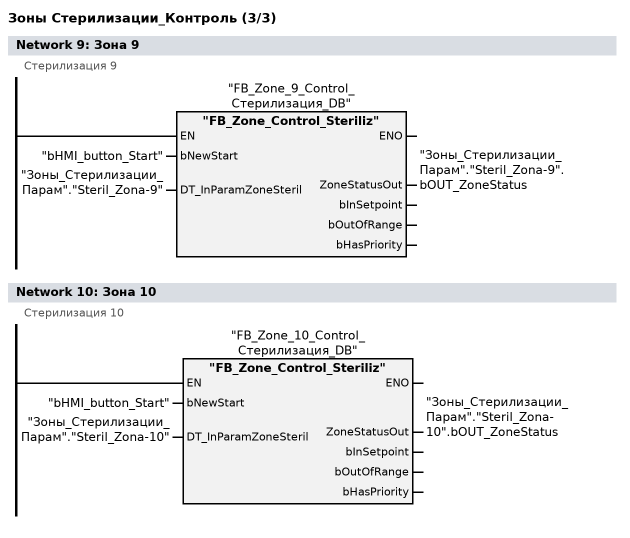
   RUNG wire#powerrail
      "FB_Zone_9_Control_Стерилизация_DB"(bNewStart := "bHMI_button_Start", DT_InParamZoneSteril := "Зоны_Стерилизации_Парам"."Steril_Zona-9", ZoneStatusOut => "Зоны_Стерилизации_Парам"."Steril_Zona-9".bOUT_ZoneStatus, bInSetpoint =>, bOutOfRange =>, bHasPriority =>)
   END_RUNG
   // the same network as SCL:
   "FB_Zone_9_Control_Стерилизация_DB"(bNewStart := "bHMI_button_Start",   // "FB_Zone_Control_Steriliz"
                           DT_InParamZoneSteril := "Зоны_Стерилизации_Парам"."Steril_Zona-9",
                           ZoneStatusOut => "Зоны_Стерилизации_Парам"."Steril_Zona-9".bOUT_ZoneStatus);
END_REGION

REGION Network 10: Зона 10
   // Стерилизация 10
   RUNG wire#powerrail
      "FB_Zone_10_Control_Стерилизация_DB"(bNewStart := "bHMI_button_Start", DT_InParamZoneSteril := "Зоны_Стерилизации_Парам"."Steril_Zona-10", ZoneStatusOut => "Зоны_Стерилизации_Парам"."Steril_Zona-10".bOUT_ZoneStatus, bInSetpoint =>, bOutOfRange =>, bHasPriority =>)
   END_RUNG
   // the same network as SCL:
   "FB_Zone_10_Control_Стерилизация_DB"(bNewStart := "bHMI_button_Start",   // "FB_Zone_Control_Steriliz"
                           DT_InParamZoneSteril := "Зоны_Стерилизации_Парам"."Steril_Zona-10",
                           ZoneStatusOut => "Зоны_Стерилизации_Парам"."Steril_Zona-10".bOUT_ZoneStatus);
END_REGION

REGION Network 11 (SCL): Соответствие выхода с датчика температур с входом для темп зоны
   "Зоны_Стерилизации_Парам"."Steril_Zona-1".rTemp := "AI_DB".AI_1.rAI_Value;
   "Зоны_Стерилизации_Парам"."Steril_Zona-2".rTemp := "AI_DB".AI_2.rAI_Value;
   "Зоны_Стерилизации_Парам"."Steril_Zona-3".rTemp := "AI_DB".AI_3.rAI_Value;
   "Зоны_Стерилизации_Парам"."Steril_Zona-4".rTemp := "AI_DB".AI_4.rAI_Value;
   "Зоны_Стерилизации_Парам"."Steril_Zona-5".rTemp := "AI_DB".AI_5.rAI_Value;
   "Зоны_Стерилизации_Парам"."Steril_Zona-6".rTemp := "AI_DB".AI_6.rAI_Value;
   "Зоны_Стерилизации_Парам"."Steril_Zona-7".rTemp := "AI_DB".AI_7.rAI_Value;
   "Зоны_Стерилизации_Парам"."Steril_Zona-8".rTemp := "AI_DB".AI_7.rAI_Value;
   "Зоны_Стерилизации_Парам"."Steril_Zona-9".rTemp := "AI_DB".AI_7.rAI_Value;
   "Зоны_Стерилизации_Парам"."Steril_Zona-10".rTemp := "AI_DB".AI_7.rAI_Value;
END_REGION
END_FUNCTION

FUNCTION "PressControl" : Void   // FC15, SCL
{ S7_Optimized_Access := 'TRUE' }
VERSION : 0.1
BEGIN

   // ---------------Присваиваем значения переменным------------------
   // 
   "Control_Press_DB".PressWater.rInPress := "AI_DB"."AI_4-20_1".rAI_Value;
   "Control_Press_DB".PressSteam.rInPress := "AI_DB"."AI_4-20_2".rAI_Value;
   "Control_Press_DB".PressGlikol.rInPress := "AI_DB"."AI_4-20_3".rAI_Value;


   //Давление ПАРА..................................................

   "FB_Press_Controll_Steam_DB"("Control_Press_DB".PressSteam);


   //Давление Воды..................................................

   "FB_Press_Controll_Water_DB"("Control_Press_DB".PressWater);


   //Давление Гликоля..................................................

   "FB_Press_Controll_Glikol_DB"("Control_Press_DB".PressGlikol);
END_FUNCTION

FUNCTION "FC_STOP" : Void   // FC16, SCL
{ S7_Optimized_Access := 'TRUE' }
VERSION : 0.1
   VAR_INPUT
      bStart : Bool;
   END_VAR
BEGIN
   IF NOT #bStart THEN
       "Pumps".Pump_1.bAutoMode_Work := False;
       "Pumps".Pump_2.bAutoMode_Work := False;
       "Pumps".Pump_3.bAutoMode_Work := False;
       "Pumps".Pump_4.bAutoMode_Work := False;
       "Pumps".Pump_5.bAutoMode_Work := False;
       "Pumps".Pump_6.bAutoMode_Work := False;
       "Pumps".Pump_7.bAutoMode_Work := False;
       "Pumps".Pump_8.bAutoMode_Work := False;
       "Pumps".Pump_9.bAutoMode_Work := False;
       "Pumps".Pump_10.bAutoMode_Work := False;




       "FVs_o/p".FV_1.bOpenCmd := FALSE;
       "FVs_o/p".FV_2.bOpenCmd := FALSE;
       "FVs_o/p".FV_3.bOpenCmd := FALSE;
       "FVs_o/p".FV_4.bOpenCmd := False;
       "FVs_o/p".FV_5.bOpenCmd := False;   

       "FVs_Regul".FV_Regul_1."bAutoOpen/Close" := FALSE;
       "FVs_Regul".FV_Regul_2."bAutoOpen/Close" := FALSE;
       "FVs_Regul".FV_Regul_3."bAutoOpen/Close" := FALSE;      //Регул клапана
       "FVs_Regul".FV_Regul_4."bAutoOpen/Close" := FALSE;
       "FVs_Regul".FV_Regul_7."bAutoOpen/Close" := FALSE;

       "bHMI_Button_ConveyorStart" := FALSE;       //Сброс кнопки подтверждения старта конвейера
       "bZoomerOff" := FALSE;

   END_IF;
END_FUNCTION

FUNCTION "Химия_насосы" : Void   // FC17, LAD
{ S7_Optimized_Access := 'TRUE' }
VERSION : 0.1
BEGIN

REGION Network 1: _____Насос Хим-1_____
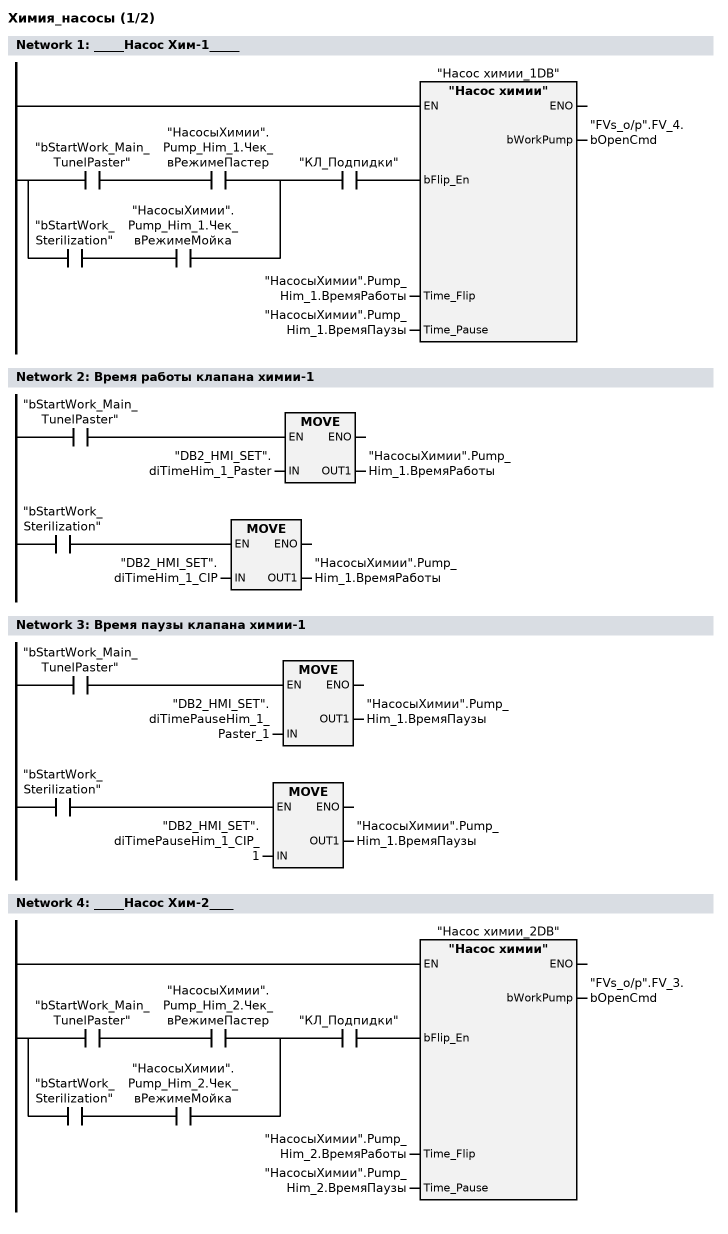
   RUNG wire#powerrail
      "Насос химии_1DB"(bFlip_En := wire#w2, Time_Flip := "НасосыХимии".Pump_Him_1.ВремяРаботы, Time_Pause := "НасосыХимии".Pump_Him_1.ВремяПаузы, bWorkPump => "FVs_o/p".FV_4.bOpenCmd)
   END_RUNG
   RUNG wire#powerrail
      Contact( "bStartWork_Main_TunelPaster" )
      Contact( "НасосыХимии".Pump_Him_1.Чек_вРежимеПастер )
      wire#w1
      Contact( "КЛ_Подпидки" )
   END_RUNG wire#w2
   RUNG wire#powerrail
      Contact( "bStartWork_Sterilization" )
      Contact( "НасосыХимии".Pump_Him_1.Чек_вРежимеМойка )
   END_RUNG wire#w1
   // the same network as SCL:
   "Насос химии_1DB"(bFlip_En := (("bStartWork_Main_TunelPaster" AND "НасосыХимии".Pump_Him_1.Чек_вРежимеПастер) OR ("bStartWork_Sterilization" AND "НасосыХимии".Pump_Him_1.Чек_вРежимеМойка)) AND "КЛ_Подпидки",   // "Насос химии"
                     Time_Flip := "НасосыХимии".Pump_Him_1.ВремяРаботы,
                     Time_Pause := "НасосыХимии".Pump_Him_1.ВремяПаузы,
                     bWorkPump => "FVs_o/p".FV_4.bOpenCmd);
END_REGION

REGION Network 2: Время работы клапана химии-1
   RUNG wire#powerrail
      Contact( "bStartWork_Main_TunelPaster" )
      Move(in := "DB2_HMI_SET".diTimeHim_1_Paster, out1 => "НасосыХимии".Pump_Him_1.ВремяРаботы)
   END_RUNG
   RUNG wire#powerrail
      Contact( "bStartWork_Sterilization" )
      Move(in := "DB2_HMI_SET".diTimeHim_1_CIP, out1 => "НасосыХимии".Pump_Him_1.ВремяРаботы)
   END_RUNG
   // the same network as SCL:
   IF "bStartWork_Main_TunelPaster" THEN
       "НасосыХимии".Pump_Him_1.ВремяРаботы := "DB2_HMI_SET".diTimeHim_1_Paster;
   END_IF;
   IF "bStartWork_Sterilization" THEN
       "НасосыХимии".Pump_Him_1.ВремяРаботы := "DB2_HMI_SET".diTimeHim_1_CIP;
   END_IF;
END_REGION

REGION Network 3: Время паузы клапана химии-1
   RUNG wire#powerrail
      Contact( "bStartWork_Main_TunelPaster" )
      Move(in := "DB2_HMI_SET".diTimePauseHim_1_Paster_1, out1 => "НасосыХимии".Pump_Him_1.ВремяПаузы)
   END_RUNG
   RUNG wire#powerrail
      Contact( "bStartWork_Sterilization" )
      Move(in := "DB2_HMI_SET".diTimePauseHim_1_CIP_1, out1 => "НасосыХимии".Pump_Him_1.ВремяПаузы)
   END_RUNG
   // the same network as SCL:
   IF "bStartWork_Main_TunelPaster" THEN
       "НасосыХимии".Pump_Him_1.ВремяПаузы := "DB2_HMI_SET".diTimePauseHim_1_Paster_1;
   END_IF;
   IF "bStartWork_Sterilization" THEN
       "НасосыХимии".Pump_Him_1.ВремяПаузы := "DB2_HMI_SET".diTimePauseHim_1_CIP_1;
   END_IF;
END_REGION

REGION Network 4: _____Насос Хим-2____
   RUNG wire#powerrail
      "Насос химии_2DB"(bFlip_En := wire#w2, Time_Flip := "НасосыХимии".Pump_Him_2.ВремяРаботы, Time_Pause := "НасосыХимии".Pump_Him_2.ВремяПаузы, bWorkPump => "FVs_o/p".FV_3.bOpenCmd)
   END_RUNG
   RUNG wire#powerrail
      Contact( "bStartWork_Main_TunelPaster" )
      Contact( "НасосыХимии".Pump_Him_2.Чек_вРежимеПастер )
      wire#w1
      Contact( "КЛ_Подпидки" )
   END_RUNG wire#w2
   RUNG wire#powerrail
      Contact( "bStartWork_Sterilization" )
      Contact( "НасосыХимии".Pump_Him_2.Чек_вРежимеМойка )
   END_RUNG wire#w1
   // the same network as SCL:
   "Насос химии_2DB"(bFlip_En := (("bStartWork_Main_TunelPaster" AND "НасосыХимии".Pump_Him_2.Чек_вРежимеПастер) OR ("bStartWork_Sterilization" AND "НасосыХимии".Pump_Him_2.Чек_вРежимеМойка)) AND "КЛ_Подпидки",   // "Насос химии"
                     Time_Flip := "НасосыХимии".Pump_Him_2.ВремяРаботы,
                     Time_Pause := "НасосыХимии".Pump_Him_2.ВремяПаузы,
                     bWorkPump => "FVs_o/p".FV_3.bOpenCmd);
END_REGION

REGION Network 5: Время работы клапана химии-2
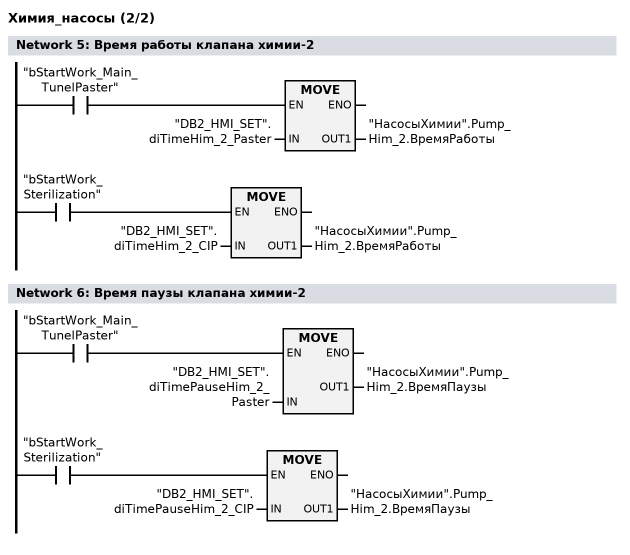
   RUNG wire#powerrail
      Contact( "bStartWork_Main_TunelPaster" )
      Move(in := "DB2_HMI_SET".diTimeHim_2_Paster, out1 => "НасосыХимии".Pump_Him_2.ВремяРаботы)
   END_RUNG
   RUNG wire#powerrail
      Contact( "bStartWork_Sterilization" )
      Move(in := "DB2_HMI_SET".diTimeHim_2_CIP, out1 => "НасосыХимии".Pump_Him_2.ВремяРаботы)
   END_RUNG
   // the same network as SCL:
   IF "bStartWork_Main_TunelPaster" THEN
       "НасосыХимии".Pump_Him_2.ВремяРаботы := "DB2_HMI_SET".diTimeHim_2_Paster;
   END_IF;
   IF "bStartWork_Sterilization" THEN
       "НасосыХимии".Pump_Him_2.ВремяРаботы := "DB2_HMI_SET".diTimeHim_2_CIP;
   END_IF;
END_REGION

REGION Network 6: Время паузы клапана химии-2
   RUNG wire#powerrail
      Contact( "bStartWork_Main_TunelPaster" )
      Move(in := "DB2_HMI_SET".diTimePauseHim_2_Paster, out1 => "НасосыХимии".Pump_Him_2.ВремяПаузы)
   END_RUNG
   RUNG wire#powerrail
      Contact( "bStartWork_Sterilization" )
      Move(in := "DB2_HMI_SET".diTimePauseHim_2_CIP, out1 => "НасосыХимии".Pump_Him_2.ВремяПаузы)
   END_RUNG
   // the same network as SCL:
   IF "bStartWork_Main_TunelPaster" THEN
       "НасосыХимии".Pump_Him_2.ВремяПаузы := "DB2_HMI_SET".diTimePauseHim_2_Paster;
   END_IF;
   IF "bStartWork_Sterilization" THEN
       "НасосыХимии".Pump_Him_2.ВремяПаузы := "DB2_HMI_SET".diTimePauseHim_2_CIP;
   END_IF;
END_REGION
END_FUNCTION

FUNCTION "Зоны БАНЯ_Контроль" : Void   // FC18, LAD
{ S7_Optimized_Access := 'TRUE' }
VERSION : 0.1
BEGIN

REGION Network 1: Зона 4
   // Зона 4
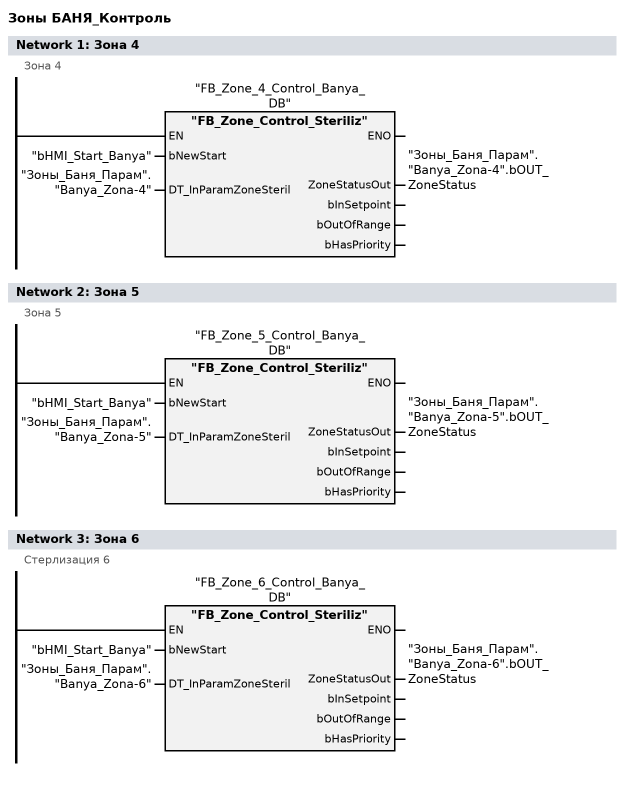
   RUNG wire#powerrail
      "FB_Zone_4_Control_Banya_DB"(bNewStart := "bHMI_Start_Banya", DT_InParamZoneSteril := "Зоны_Баня_Парам"."Banya_Zona-4", ZoneStatusOut => "Зоны_Баня_Парам"."Banya_Zona-4".bOUT_ZoneStatus, bInSetpoint =>, bOutOfRange =>, bHasPriority =>)
   END_RUNG
   // the same network as SCL:
   "FB_Zone_4_Control_Banya_DB"(bNewStart := "bHMI_Start_Banya",   // "FB_Zone_Control_Steriliz"
                           DT_InParamZoneSteril := "Зоны_Баня_Парам"."Banya_Zona-4",
                           ZoneStatusOut => "Зоны_Баня_Парам"."Banya_Zona-4".bOUT_ZoneStatus);
END_REGION

REGION Network 2: Зона 5
   // Зона 5
   RUNG wire#powerrail
      "FB_Zone_5_Control_Banya_DB"(bNewStart := "bHMI_Start_Banya", DT_InParamZoneSteril := "Зоны_Баня_Парам"."Banya_Zona-5", ZoneStatusOut => "Зоны_Баня_Парам"."Banya_Zona-5".bOUT_ZoneStatus, bInSetpoint =>, bOutOfRange =>, bHasPriority =>)
   END_RUNG
   // the same network as SCL:
   "FB_Zone_5_Control_Banya_DB"(bNewStart := "bHMI_Start_Banya",   // "FB_Zone_Control_Steriliz"
                           DT_InParamZoneSteril := "Зоны_Баня_Парам"."Banya_Zona-5",
                           ZoneStatusOut => "Зоны_Баня_Парам"."Banya_Zona-5".bOUT_ZoneStatus);
END_REGION

REGION Network 3: Зона 6
   // Стерлизация 6
   RUNG wire#powerrail
      "FB_Zone_6_Control_Banya_DB"(bNewStart := "bHMI_Start_Banya", DT_InParamZoneSteril := "Зоны_Баня_Парам"."Banya_Zona-6", ZoneStatusOut => "Зоны_Баня_Парам"."Banya_Zona-6".bOUT_ZoneStatus, bInSetpoint =>, bOutOfRange =>, bHasPriority =>)
   END_RUNG
   // the same network as SCL:
   "FB_Zone_6_Control_Banya_DB"(bNewStart := "bHMI_Start_Banya",   // "FB_Zone_Control_Steriliz"
                           DT_InParamZoneSteril := "Зоны_Баня_Парам"."Banya_Zona-6",
                           ZoneStatusOut => "Зоны_Баня_Парам"."Banya_Zona-6".bOUT_ZoneStatus);
END_REGION

REGION Network 4 (SCL): Соответствие выхода с датчика температур с входом для темп зоны
   "Зоны_Стерилизации_Парам"."Steril_Zona-1".rTemp := "AI_DB".AI_1.rAI_Value;
   "Зоны_Стерилизации_Парам"."Steril_Zona-2".rTemp := "AI_DB".AI_2.rAI_Value;
   "Зоны_Стерилизации_Парам"."Steril_Zona-3".rTemp := "AI_DB".AI_3.rAI_Value;
   "Зоны_Стерилизации_Парам"."Steril_Zona-4".rTemp := "AI_DB".AI_4.rAI_Value;
   "Зоны_Стерилизации_Парам"."Steril_Zona-5".rTemp := "AI_DB".AI_5.rAI_Value;
   "Зоны_Стерилизации_Парам"."Steril_Zona-6".rTemp := "AI_DB".AI_6.rAI_Value;
   "Зоны_Стерилизации_Парам"."Steril_Zona-7".rTemp := "AI_DB".AI_7.rAI_Value;
   "Зоны_Стерилизации_Парам"."Steril_Zona-8".rTemp := "AI_DB".AI_7.rAI_Value;
   "Зоны_Стерилизации_Парам"."Steril_Zona-9".rTemp := "AI_DB".AI_7.rAI_Value;
   "Зоны_Стерилизации_Парам"."Steril_Zona-10".rTemp := "AI_DB".AI_7.rAI_Value;
END_REGION
END_FUNCTION

ORGANIZATION_BLOCK "Main"   // OB1, LAD, ProgramCycle
TITLE = "Основкая программа"
{ S7_Optimized_Access := 'TRUE' }
VERSION : 0.1
   VAR_TEMP
      Off : Bool;
   END_VAR
BEGIN

REGION Network 1: Аварии
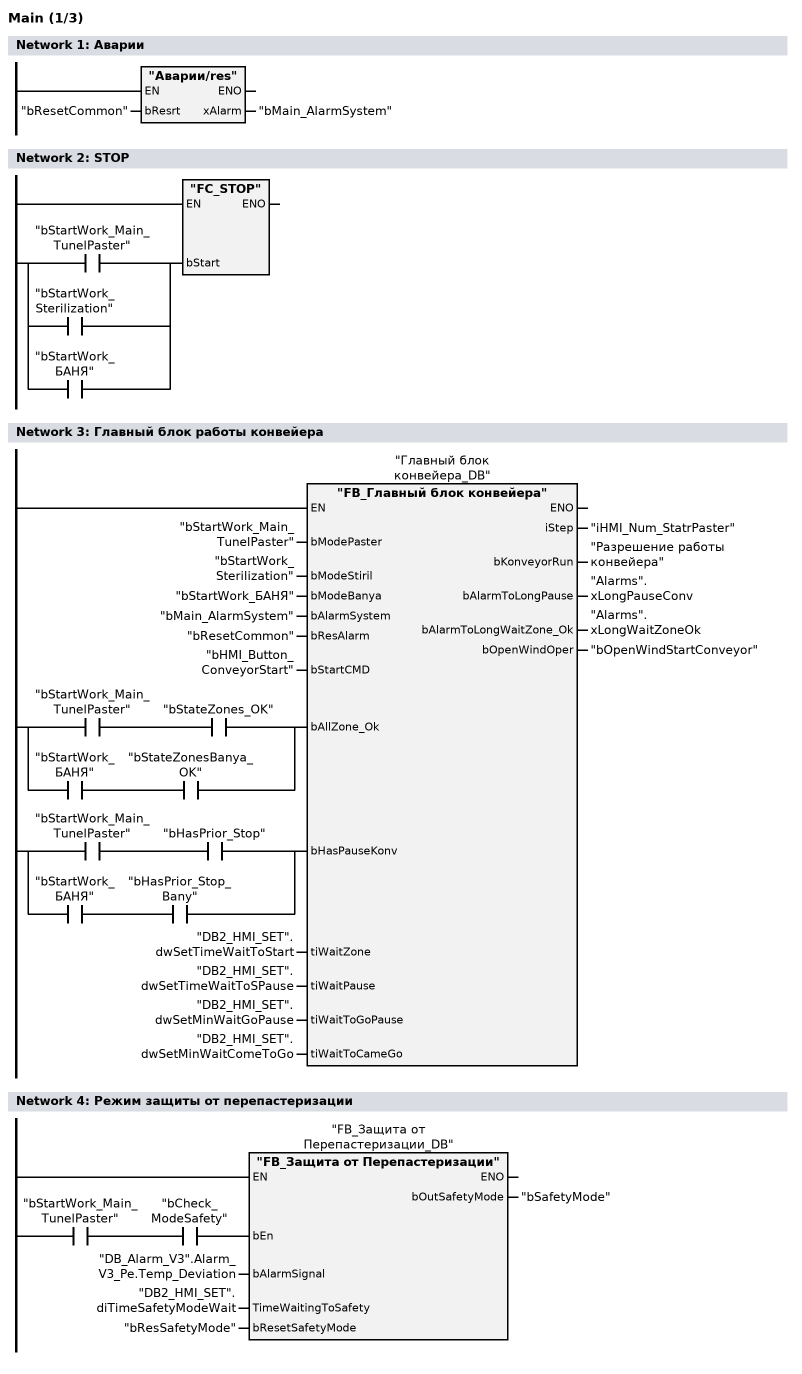
   RUNG wire#powerrail
      "Аварии/res"(bResrt := "bResetCommon", xAlarm => "bMain_AlarmSystem")
   END_RUNG
   // the same network as SCL:
   "Аварии/res"(bResrt := "bResetCommon", xAlarm => "bMain_AlarmSystem");
END_REGION

REGION Network 2: STOP
   RUNG wire#powerrail
      "FC_STOP"(bStart := wire#w1)
   END_RUNG
   RUNG wire#powerrail
      Contact( "bStartWork_Main_TunelPaster" )
   END_RUNG wire#w1
   RUNG wire#powerrail
      Contact( "bStartWork_Sterilization" )
   END_RUNG wire#w1
   RUNG wire#powerrail
      Contact( "bStartWork_БАНЯ" )
   END_RUNG wire#w1
   // the same network as SCL:
   "FC_STOP"(bStart := "bStartWork_Main_TunelPaster" OR "bStartWork_Sterilization" OR "bStartWork_БАНЯ");
END_REGION

REGION Network 3: Главный блок работы конвейера
   RUNG wire#powerrail
      "Главный блок конвейера_DB"(bAllZone_Ok := wire#w1, bHasPauseKonv := wire#w2, bModePaster := "bStartWork_Main_TunelPaster", bModeStiril := "bStartWork_Sterilization", bModeBanya := "bStartWork_БАНЯ", bAlarmSystem := "bMain_AlarmSystem", bResAlarm := "bResetCommon", bStartCMD := "bHMI_Button_ConveyorStart", tiWaitZone := "DB2_HMI_SET".dwSetTimeWaitToStart, tiWaitPause := "DB2_HMI_SET".dwSetTimeWaitToSPause, tiWaitToGoPause := "DB2_HMI_SET".dwSetMinWaitGoPause, tiWaitToCameGo := "DB2_HMI_SET".dwSetMinWaitComeToGo, iStep => "iHMI_Num_StatrPaster", bKonveyorRun => "Разрешение работы конвейера", bAlarmToLongPause => "Alarms".xLongPauseConv, bAlarmToLongWaitZone_Ok => "Alarms".xLongWaitZoneOk, bOpenWindOper => "bOpenWindStartConveyor")
   END_RUNG
   RUNG wire#powerrail
      Contact( "bStartWork_Main_TunelPaster" )
      Contact( "bStateZones_OK" )
   END_RUNG wire#w1
   RUNG wire#powerrail
      Contact( "bStartWork_БАНЯ" )
      Contact( "bStateZonesBanya_OK" )
   END_RUNG wire#w1
   RUNG wire#powerrail
      Contact( "bStartWork_Main_TunelPaster" )
      Contact( "bHasPrior_Stop" )
   END_RUNG wire#w2
   RUNG wire#powerrail
      Contact( "bStartWork_БАНЯ" )
      Contact( "bHasPrior_Stop_Bany" )
   END_RUNG wire#w2
   // the same network as SCL:
   "Главный блок конвейера_DB"(bModePaster := "bStartWork_Main_TunelPaster",   // "FB_Главный блок конвейера"
                           bModeStiril := "bStartWork_Sterilization",
                           bModeBanya := "bStartWork_БАНЯ",
                           bAlarmSystem := "bMain_AlarmSystem",
                           bResAlarm := "bResetCommon",
                           bStartCMD := "bHMI_Button_ConveyorStart",
                           bAllZone_Ok := ("bStartWork_Main_TunelPaster" AND "bStateZones_OK") OR ("bStartWork_БАНЯ" AND "bStateZonesBanya_OK"),
                           bHasPauseKonv := ("bStartWork_Main_TunelPaster" AND "bHasPrior_Stop") OR ("bStartWork_БАНЯ" AND "bHasPrior_Stop_Bany"),
                           tiWaitZone := "DB2_HMI_SET".dwSetTimeWaitToStart,
                           tiWaitPause := "DB2_HMI_SET".dwSetTimeWaitToSPause,
                           tiWaitToGoPause := "DB2_HMI_SET".dwSetMinWaitGoPause,
                           tiWaitToCameGo := "DB2_HMI_SET".dwSetMinWaitComeToGo,
                           iStep => "iHMI_Num_StatrPaster",
                           bKonveyorRun => "Разрешение работы конвейера",
                           bAlarmToLongPause => "Alarms".xLongPauseConv,
                           bAlarmToLongWaitZone_Ok => "Alarms".xLongWaitZoneOk,
                           bOpenWindOper => "bOpenWindStartConveyor");
END_REGION

REGION Network 4: Режим защиты от перепастеризации
   RUNG wire#powerrail
      "FB_Защита от Перепастеризации_DB"(bEn := wire#w1, bAlarmSignal := "DB_Alarm_V3".Alarm_V3_Pe.Temp_Deviation, TimeWaitingToSafety := "DB2_HMI_SET".diTimeSafetyModeWait, bResetSafetyMode := "bResSafetyMode", bOutSafetyMode => "bSafetyMode")
   END_RUNG
   RUNG wire#powerrail
      Contact( "bStartWork_Main_TunelPaster" )
      Contact( "bCheck_ModeSafety" )
   END_RUNG wire#w1
   // the same network as SCL:
   "FB_Защита от Перепастеризации_DB"(bEn := "bStartWork_Main_TunelPaster" AND "bCheck_ModeSafety",   // "FB_Защита от Перепастеризации"
                           bAlarmSignal := "DB_Alarm_V3".Alarm_V3_Pe.Temp_Deviation,
                           TimeWaitingToSafety := "DB2_HMI_SET".diTimeSafetyModeWait,
                           bResetSafetyMode := "bResSafetyMode",
                           bOutSafetyMode => "bSafetyMode");
END_REGION

REGION Network 5: Расчет PE и скорости конвейера (Верс-1)
   // Блок работы расчета ПЕ и скорости - скорость считается по параметрам частотника
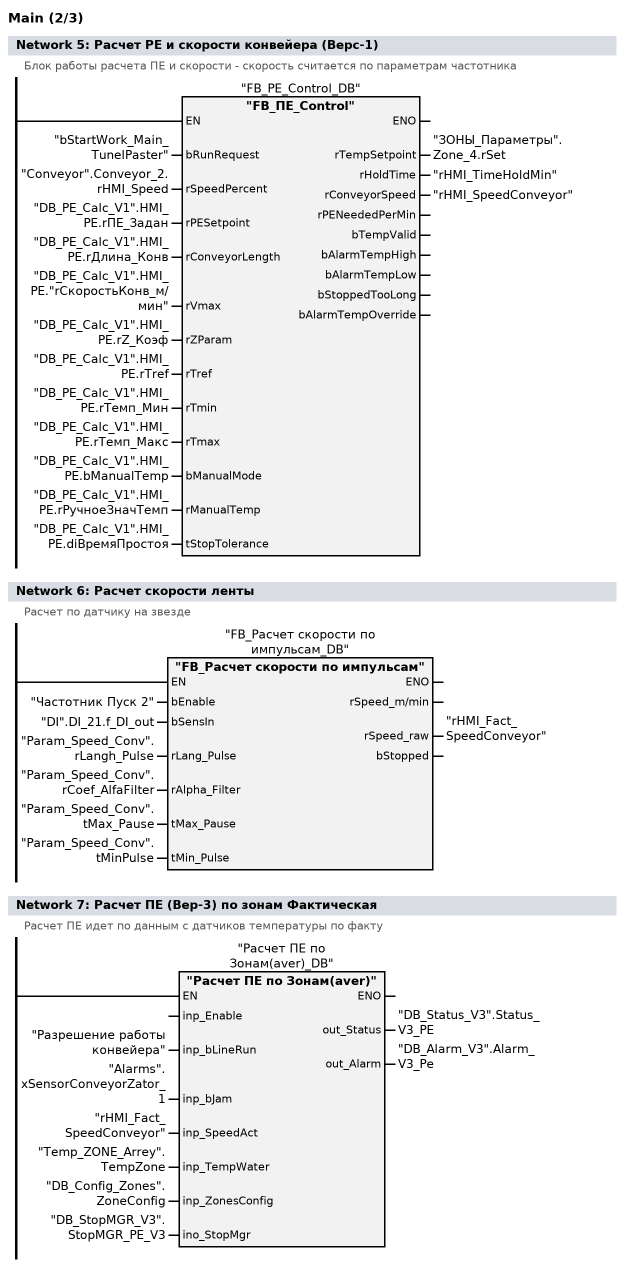
   RUNG wire#powerrail
      "FB_PE_Control_DB"(bRunRequest := "bStartWork_Main_TunelPaster", rSpeedPercent := "Conveyor".Conveyor_2.rHMI_Speed, rPESetpoint := "DB_PE_Calc_V1".HMI_PE.rПЕ_Задан, rConveyorLength := "DB_PE_Calc_V1".HMI_PE.rДлина_Конв, rVmax := "DB_PE_Calc_V1".HMI_PE."rСкоростьКонв_м/мин", rZParam := "DB_PE_Calc_V1".HMI_PE.rZ_Коэф, rTref := "DB_PE_Calc_V1".HMI_PE.rТref, rTmin := "DB_PE_Calc_V1".HMI_PE.rТемп_Мин, rTmax := "DB_PE_Calc_V1".HMI_PE.rТемп_Макс, bManualMode := "DB_PE_Calc_V1".HMI_PE.bManualTemp, rManualTemp := "DB_PE_Calc_V1".HMI_PE.rРучноеЗначТемп, tStopTolerance := "DB_PE_Calc_V1".HMI_PE.diВремяПростоя, rTempSetpoint => "ЗОНЫ_Параметры".Zone_4.rSet, rHoldTime => "rHMI_TimeHoldMin", rConveyorSpeed => "rHMI_SpeedConveyor", rPENeededPerMin =>, bTempValid =>, bAlarmTempHigh =>, bAlarmTempLow =>, bStoppedTooLong =>, bAlarmTempOverride =>)
   END_RUNG
   // the same network as SCL:
   "FB_PE_Control_DB"(bRunRequest := "bStartWork_Main_TunelPaster",   // "FB_ПЕ_Control"
                      rSpeedPercent := "Conveyor".Conveyor_2.rHMI_Speed,
                      rPESetpoint := "DB_PE_Calc_V1".HMI_PE.rПЕ_Задан,
                      rConveyorLength := "DB_PE_Calc_V1".HMI_PE.rДлина_Конв,
                      rVmax := "DB_PE_Calc_V1".HMI_PE."rСкоростьКонв_м/мин",
                      rZParam := "DB_PE_Calc_V1".HMI_PE.rZ_Коэф,
                      rTref := "DB_PE_Calc_V1".HMI_PE.rТref,
                      rTmin := "DB_PE_Calc_V1".HMI_PE.rТемп_Мин,
                      rTmax := "DB_PE_Calc_V1".HMI_PE.rТемп_Макс,
                      bManualMode := "DB_PE_Calc_V1".HMI_PE.bManualTemp,
                      rManualTemp := "DB_PE_Calc_V1".HMI_PE.rРучноеЗначТемп,
                      tStopTolerance := "DB_PE_Calc_V1".HMI_PE.diВремяПростоя,
                      rTempSetpoint => "ЗОНЫ_Параметры".Zone_4.rSet,
                      rHoldTime => "rHMI_TimeHoldMin",
                      rConveyorSpeed => "rHMI_SpeedConveyor");
END_REGION

REGION Network 6: Расчет скорости ленты
   // Расчет по датчику на звезде
   RUNG wire#powerrail
      "FB_Расчет скорости по импульсам_DB"(bEnable := "Частотник Пуск 2", bSensIn := "DI".DI_21.f_DI_out, rLang_Pulse := "Param_Speed_Conv".rLangh_Pulse, rAlpha_Filter := "Param_Speed_Conv".rCoef_AlfaFilter, tMax_Pause := "Param_Speed_Conv".tMax_Pause, tMin_Pulse := "Param_Speed_Conv".tMinPulse, "rSpeed_m/min" =>, rSpeed_raw => "rHMI_Fact_SpeedConveyor", bStopped =>)
   END_RUNG
   // the same network as SCL:
   "FB_Расчет скорости по импульсам_DB"(bEnable := "Частотник Пуск 2",   // "FB_Расчет скорости по импульсам"
                           bSensIn := "DI".DI_21.f_DI_out,
                           rLang_Pulse := "Param_Speed_Conv".rLangh_Pulse,
                           rAlpha_Filter := "Param_Speed_Conv".rCoef_AlfaFilter,
                           tMax_Pause := "Param_Speed_Conv".tMax_Pause,
                           tMin_Pulse := "Param_Speed_Conv".tMinPulse,
                           rSpeed_raw => "rHMI_Fact_SpeedConveyor");
END_REGION

REGION Network 7: Расчет ПЕ (Вер-3) по зонам Фактическая
   // Расчет ПЕ идет по данным с датчиков температуры по факту
   RUNG wire#powerrail
      "Расчет ПЕ по Зонам(aver)_DB"(inp_Enable :=, inp_bLineRun := "Разрешение работы конвейера", inp_bJam := "Alarms".xSensorConveyorZator_1, inp_SpeedAct := "rHMI_Fact_SpeedConveyor", inp_TempWater := "Temp_ZONE_Arrey".TempZone, inp_ZonesConfig := "DB_Config_Zones".ZoneConfig, ino_StopMgr := "DB_StopMGR_V3".StopMGR_PE_V3, out_Status => "DB_Status_V3".Status_V3_PE, out_Alarm => "DB_Alarm_V3".Alarm_V3_Pe)
   END_RUNG
   // the same network as SCL:
   "Расчет ПЕ по Зонам(aver)_DB"(inp_bLineRun := "Разрешение работы конвейера",   // "Расчет ПЕ по Зонам(aver)"
                           inp_bJam := "Alarms".xSensorConveyorZator_1,
                           inp_SpeedAct := "rHMI_Fact_SpeedConveyor",
                           inp_TempWater := "Temp_ZONE_Arrey".TempZone,
                           inp_ZonesConfig := "DB_Config_Zones".ZoneConfig,
                           ino_StopMgr := "DB_StopMGR_V3".StopMGR_PE_V3,
                           out_Status => "DB_Status_V3".Status_V3_PE,
                           out_Alarm => "DB_Alarm_V3".Alarm_V3_Pe);
END_REGION

REGION Network 8 (SCL): Температуры по зонам в массив
   // Перевод значений температур воды по зонам в массив для использования в блоке
   //============== Фактическая температура =========================
   "Temp_ZONE_Arrey".TempZone[1] := "ЗОНЫ_Параметры".Zone_1.rTemp;
   "Temp_ZONE_Arrey".TempZone[2] := "ЗОНЫ_Параметры".Zone_2.rTemp;
   "Temp_ZONE_Arrey".TempZone[3] := "ЗОНЫ_Параметры".Zone_3.rTemp;
   "Temp_ZONE_Arrey".TempZone[4] := "ЗОНЫ_Параметры".Zone_4.rTemp;
   "Temp_ZONE_Arrey".TempZone[5] := "ЗОНЫ_Параметры".Zone_5.rTemp;
   "Temp_ZONE_Arrey".TempZone[6] := "ЗОНЫ_Параметры".Zone_6.rTemp;
   "Temp_ZONE_Arrey".TempZone[7] := "ЗОНЫ_Параметры".Zone_7.rTemp;
   "Temp_ZONE_Arrey".TempZone[8] := "ЗОНЫ_Параметры".Zone_8.rTemp;
   "Temp_ZONE_Arrey".TempZone[9] := "ЗОНЫ_Параметры".Zone_9.rTemp;
   //============== Уставка температур ====================================
   "DB_Config_Zones".ZoneConfig[1].TempWater_Set:= "ЗОНЫ_Параметры".Zone_1.rSet;
   "DB_Config_Zones".ZoneConfig[2].TempWater_Set := "ЗОНЫ_Параметры".Zone_2.rSet;
   "DB_Config_Zones".ZoneConfig[3].TempWater_Set := "ЗОНЫ_Параметры".Zone_3.rSet;
   "DB_Config_Zones".ZoneConfig[4].TempWater_Set := "ЗОНЫ_Параметры".Zone_4.rSet;
   "DB_Config_Zones".ZoneConfig[5].TempWater_Set := "ЗОНЫ_Параметры".Zone_5.rSet;
   "DB_Config_Zones".ZoneConfig[6].TempWater_Set := "ЗОНЫ_Параметры".Zone_6.rSet;
   "DB_Config_Zones".ZoneConfig[7].TempWater_Set := "ЗОНЫ_Параметры".Zone_7.rSet;
   "DB_Config_Zones".ZoneConfig[8].TempWater_Set := "ЗОНЫ_Параметры".Zone_8.rSet;
   "DB_Config_Zones".ZoneConfig[9].TempWater_Set := "ЗОНЫ_Параметры".Zone_9.rSet;
END_REGION

REGION Network 9: Расчет ПЕ (Вер-3) по зонам - РАСЧЕТНАЯ
   // Расчетное значение ПЕ считается по утсавкам температур в зонах - для расчетной берем уставку и подстваляем под значение температуры в зоне - получается идеальный вариант температур и сколько буде ПЕ при идеальных условиях
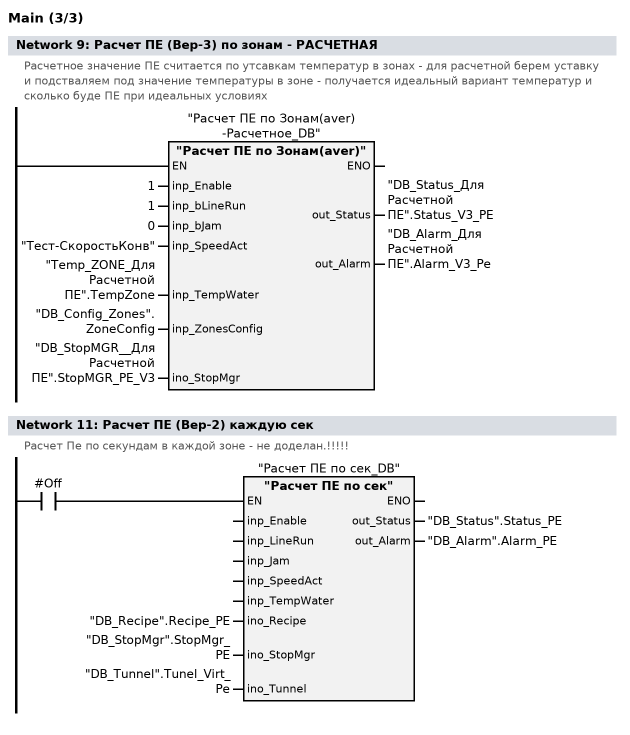
   RUNG wire#powerrail
      "Расчет ПЕ по Зонам(aver) -Расчетное_DB"(inp_Enable := 1, inp_bLineRun := 1, inp_bJam := 0, inp_SpeedAct := "Тест-СкоростьКонв", inp_TempWater := "Temp_ZONE_Для Расчетной ПЕ".TempZone, inp_ZonesConfig := "DB_Config_Zones".ZoneConfig, ino_StopMgr := "DB_StopMGR__Для Расчетной ПЕ".StopMGR_PE_V3, out_Status => "DB_Status_Для Расчетной ПЕ".Status_V3_PE, out_Alarm => "DB_Alarm_Для Расчетной ПЕ".Alarm_V3_Pe)
   END_RUNG
   // the same network as SCL:
   "Расчет ПЕ по Зонам(aver) -Расчетное_DB"(inp_Enable := 1,   // "Расчет ПЕ по Зонам(aver)"
                           inp_bLineRun := 1,
                           inp_bJam := 0,
                           inp_SpeedAct := "Тест-СкоростьКонв",
                           inp_TempWater := "Temp_ZONE_Для Расчетной ПЕ".TempZone,
                           inp_ZonesConfig := "DB_Config_Zones".ZoneConfig,
                           ino_StopMgr := "DB_StopMGR__Для Расчетной ПЕ".StopMGR_PE_V3,
                           out_Status => "DB_Status_Для Расчетной ПЕ".Status_V3_PE,
                           out_Alarm => "DB_Alarm_Для Расчетной ПЕ".Alarm_V3_Pe);
END_REGION

REGION Network 10 (SCL): Температуры по зонам в массив - РАСЧЕТНАЯ
   // Перевод значений температур воды по зонам в массив для использования в блоке
   //============== Фактическая температура =========================
   "Temp_ZONE_Для Расчетной ПЕ".TempZone[1] := "ЗОНЫ_Параметры".Zone_1.rSet;
   "Temp_ZONE_Для Расчетной ПЕ".TempZone[2] := "ЗОНЫ_Параметры".Zone_2.rSet;
   "Temp_ZONE_Для Расчетной ПЕ".TempZone[3] := "ЗОНЫ_Параметры".Zone_3.rSet;
   "Temp_ZONE_Для Расчетной ПЕ".TempZone[4] := "ЗОНЫ_Параметры".Zone_4.rSet;
   "Temp_ZONE_Для Расчетной ПЕ".TempZone[5] := "ЗОНЫ_Параметры".Zone_5.rSet;
   "Temp_ZONE_Для Расчетной ПЕ".TempZone[6] := "ЗОНЫ_Параметры".Zone_6.rSet;
   "Temp_ZONE_Для Расчетной ПЕ".TempZone[7] := "ЗОНЫ_Параметры".Zone_7.rSet;
   "Temp_ZONE_Для Расчетной ПЕ".TempZone[8] := "ЗОНЫ_Параметры".Zone_8.rSet;
   "Temp_ZONE_Для Расчетной ПЕ".TempZone[9] := "ЗОНЫ_Параметры".Zone_9.rSet;
   //============== Уставка температур ====================================
   "DB_Config_Zones".ZoneConfig[1].TempWater_Set := "ЗОНЫ_Параметры".Zone_1.rSet;
   "DB_Config_Zones".ZoneConfig[2].TempWater_Set := "ЗОНЫ_Параметры".Zone_2.rSet;
   "DB_Config_Zones".ZoneConfig[3].TempWater_Set := "ЗОНЫ_Параметры".Zone_3.rSet;
   "DB_Config_Zones".ZoneConfig[4].TempWater_Set := "ЗОНЫ_Параметры".Zone_4.rSet;
   "DB_Config_Zones".ZoneConfig[5].TempWater_Set := "ЗОНЫ_Параметры".Zone_5.rSet;
   "DB_Config_Zones".ZoneConfig[6].TempWater_Set := "ЗОНЫ_Параметры".Zone_6.rSet;
   "DB_Config_Zones".ZoneConfig[7].TempWater_Set := "ЗОНЫ_Параметры".Zone_7.rSet;
   "DB_Config_Zones".ZoneConfig[8].TempWater_Set := "ЗОНЫ_Параметры".Zone_8.rSet;
   "DB_Config_Zones".ZoneConfig[9].TempWater_Set := "ЗОНЫ_Параметры".Zone_9.rSet;
END_REGION

REGION Network 11: Расчет ПЕ (Вер-2) каждую сек
   // Расчет Пе по секундам в каждой зоне - не доделан.!!!!!
   RUNG wire#powerrail
      Contact( #Off )
      "Расчет ПЕ по сек_DB"(inp_Enable :=, inp_LineRun :=, inp_Jam :=, inp_SpeedAct :=, inp_TempWater :=, ino_Recipe := "DB_Recipe".Recipe_PE, ino_StopMgr := "DB_StopMgr".StopMgr_PE, ino_Tunnel := "DB_Tunnel".Tunel_Virt_Pe, out_Status => "DB_Status".Status_PE, out_Alarm => "DB_Alarm".Alarm_PE)
   END_RUNG
   // the same network as SCL:
   IF #Off THEN
       "Расчет ПЕ по сек_DB"(ino_Recipe := "DB_Recipe".Recipe_PE,   // "Расчет ПЕ по сек"
                             ino_StopMgr := "DB_StopMgr".StopMgr_PE,
                             ino_Tunnel := "DB_Tunnel".Tunel_Virt_Pe,
                             out_Status => "DB_Status".Status_PE,
                             out_Alarm => "DB_Alarm".Alarm_PE);
   END_IF;
END_REGION
END_ORGANIZATION_BLOCK

ORGANIZATION_BLOCK "PID"   // OB30, LAD, CyclicInterrupt
{ S7_Optimized_Access := 'TRUE' }
VERSION : 0.1
   VAR_INPUT
      Initial_Call : Bool;   // Initial call of this OB
      Event_Count : Int;   // Events discarded
   END_VAR
BEGIN

REGION Network 1: ПИД - Зона 1
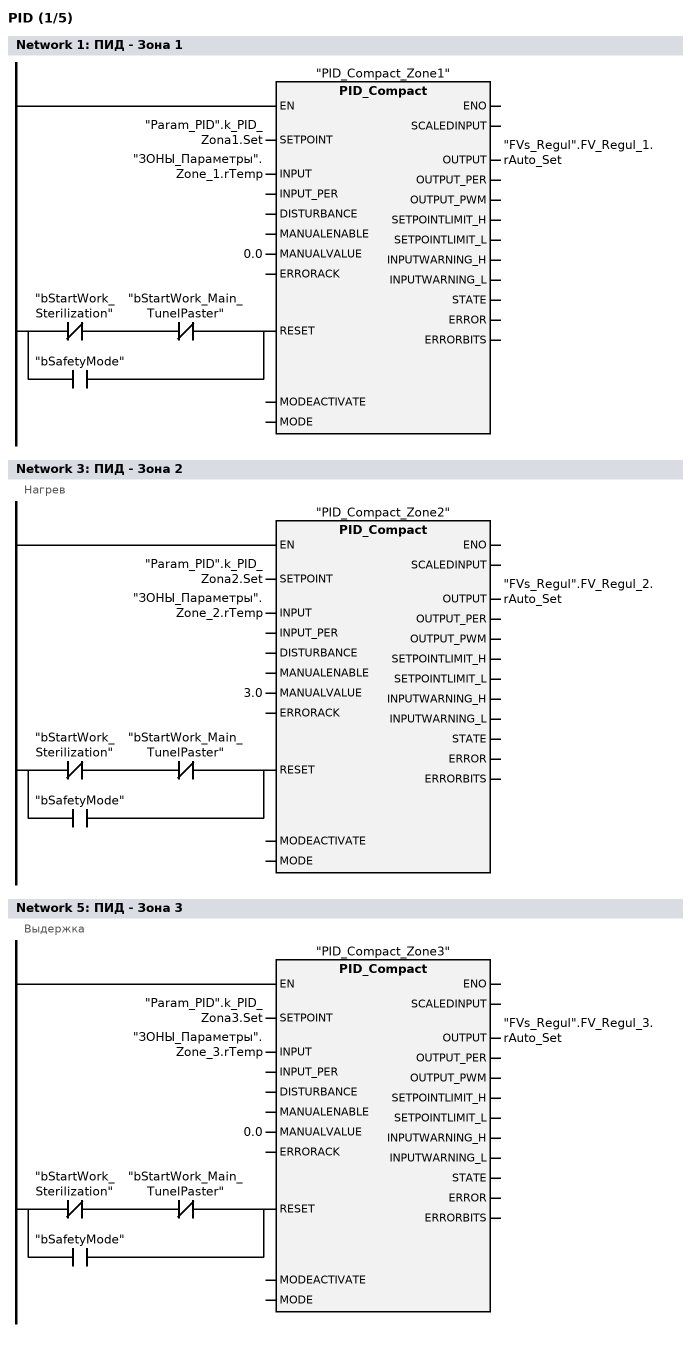
   "PID_Compact_Zone1"(Setpoint := "Param_PID".k_PID_Zona1.Set,   // PID_Compact
                       Input := "ЗОНЫ_Параметры".Zone_1.rTemp,
                       ManualValue := 0.0,
                       Reset := (NOT "bStartWork_Sterilization" AND NOT "bStartWork_Main_TunelPaster") OR "bSafetyMode",
                       Output => "FVs_Regul".FV_Regul_1.rAuto_Set);
END_REGION

REGION Network 2 (SCL): Выбор типа ПИД - Зона 1
   //Режим работы ПИД - 0 - Нагрев; 1 - Охлаждение
   "PID_Compact_Zone1".Config.InvertControl := "bTypePID_Zone1";
   //Задание коэффициэнтов в ручном режиме

   "PID_Compact_Zone1".Retain.CtrlParams.Gain := "Param_PID".k_PID_Zona1.Gain; // Изменение коэф. П
   "PID_Compact_Zone1".Retain.CtrlParams.Ti  := "Param_PID".k_PID_Zona1.I; // Изменение коэф И
   "PID_Compact_Zone1".Retain.CtrlParams.Td  := "Param_PID".k_PID_Zona1.D; // Изменение коэф Д
END_REGION

REGION Network 3: ПИД - Зона 2
   // Нагрев
   "PID_Compact_Zone2"(Setpoint := "Param_PID".k_PID_Zona2.Set,   // PID_Compact
                       Input := "ЗОНЫ_Параметры".Zone_2.rTemp,
                       ManualValue := 3.0,
                       Reset := (NOT "bStartWork_Sterilization" AND NOT "bStartWork_Main_TunelPaster") OR "bSafetyMode",
                       Output => "FVs_Regul".FV_Regul_2.rAuto_Set);
END_REGION

REGION Network 4 (SCL): Выбор типа ПИД Зона 2
   // 0 - Нагрев; 1 - Охлаждение
   //Режим работы ПИД - 0 - Нагрев; 1 - Охлаждение
   "PID_Compact_Zone2".Config.InvertControl := "bTypePID_Zone2";
   //Задание коэффициэнтов в ручном режиме

   "PID_Compact_Zone2".Retain.CtrlParams.Gain := "Param_PID".k_PID_Zona2.Gain; // Изменение коэф. П
   "PID_Compact_Zone2".Retain.CtrlParams.Ti := "Param_PID".k_PID_Zona2.I; // Изменение коэф И
   "PID_Compact_Zone2".Retain.CtrlParams.Td := "Param_PID".k_PID_Zona2.D; // Изменение коэф Д
END_REGION

REGION Network 5: ПИД - Зона 3
   // Выдержка
   "PID_Compact_Zone3"(Setpoint := "Param_PID".k_PID_Zona3.Set,   // PID_Compact
                       Input := "ЗОНЫ_Параметры".Zone_3.rTemp,
                       ManualValue := 0.0,
                       Reset := (NOT "bStartWork_Sterilization" AND NOT "bStartWork_Main_TunelPaster") OR "bSafetyMode",
                       Output => "FVs_Regul".FV_Regul_3.rAuto_Set);
END_REGION

REGION Network 6 (SCL): Выбор типа ПИД Зона 3
   // 0 - Нагрев; 1 - Охлаждение
   //Режим работы ПИД - 0 - Нагрев; 1 - Охлаждение
   "PID_Compact_Zone3".Config.InvertControl := "bTypePID_Zone3";
   //Задание коэффициэнтов в ручном режиме

   "PID_Compact_Zone3".Retain.CtrlParams.Gain := "Param_PID".k_PID_Zona3.Gain; // Изменение коэф. П
   "PID_Compact_Zone3".Retain.CtrlParams.Ti := "Param_PID".k_PID_Zona3.I; // Изменение коэф И
   "PID_Compact_Zone3".Retain.CtrlParams.Td := "Param_PID".k_PID_Zona3.D; // Изменение коэф Д
END_REGION

REGION Network 7: ПИД - Зона 4
   // Выдержка
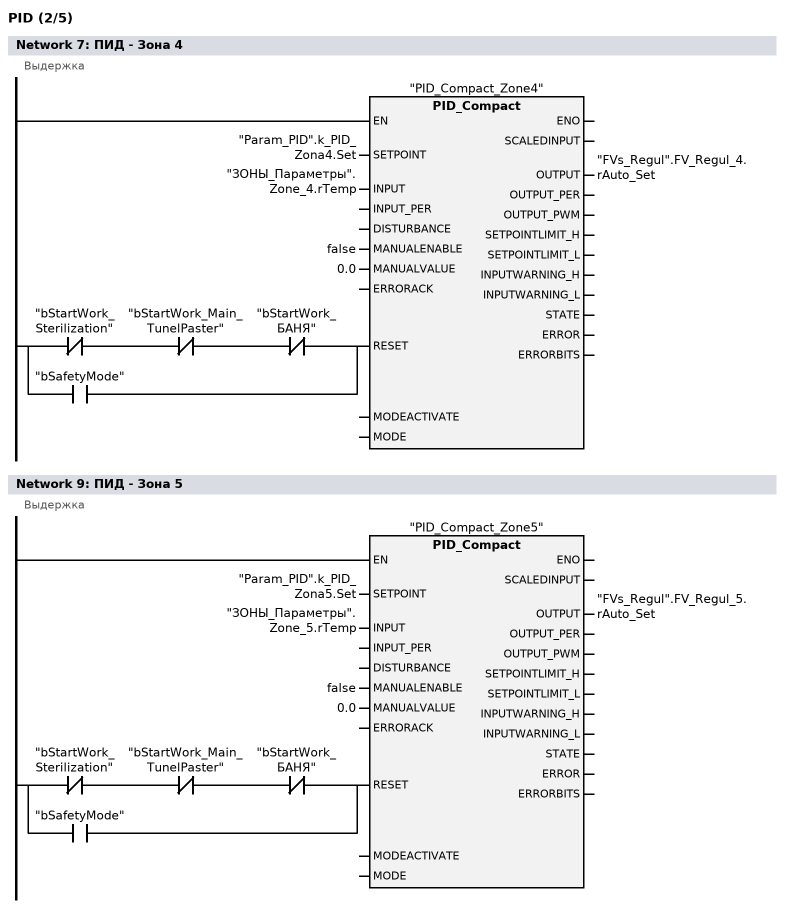
   "PID_Compact_Zone4"(Setpoint := "Param_PID".k_PID_Zona4.Set,   // PID_Compact
                       Input := "ЗОНЫ_Параметры".Zone_4.rTemp,
                       ManualEnable := false,
                       ManualValue := 0.0,
                       Reset := (NOT "bStartWork_Sterilization" AND NOT "bStartWork_Main_TunelPaster" AND NOT "bStartWork_БАНЯ") OR "bSafetyMode",
                       Output => "FVs_Regul".FV_Regul_4.rAuto_Set);
END_REGION

REGION Network 8 (SCL): Выбор типа ПИД Зона 4
   // 0 - Нагрев; 1 - Охлаждение
   //Режим работы ПИД - 0 - Нагрев; 1 - Охлаждение
   "PID_Compact_Zone4".Config.InvertControl := "bTypePID_Zone4";
   //Задание коэффициэнтов в ручном режиме

   "PID_Compact_Zone4".Retain.CtrlParams.Gain := "Param_PID".k_PID_Zona4.Gain; // Изменение коэф. П
   "PID_Compact_Zone4".Retain.CtrlParams.Ti := "Param_PID".k_PID_Zona4.I; // Изменение коэф И
   "PID_Compact_Zone4".Retain.CtrlParams.Td := "Param_PID".k_PID_Zona4.D; // Изменение коэф Д
END_REGION

REGION Network 9: ПИД - Зона 5
   // Выдержка
   "PID_Compact_Zone5"(Setpoint := "Param_PID".k_PID_Zona5.Set,   // PID_Compact
                       Input := "ЗОНЫ_Параметры".Zone_5.rTemp,
                       ManualEnable := false,
                       ManualValue := 0.0,
                       Reset := (NOT "bStartWork_Sterilization" AND NOT "bStartWork_Main_TunelPaster" AND NOT "bStartWork_БАНЯ") OR "bSafetyMode",
                       Output => "FVs_Regul".FV_Regul_5.rAuto_Set);
END_REGION

REGION Network 10 (SCL): Выбор типа ПИД Зона 5
   // 0 - Нагрев; 1 - Охлаждение
   //Режим работы ПИД - 0 - Нагрев; 1 - Охлаждение
   "PID_Compact_Zone5".Config.InvertControl := "bTypePID_Zone5";
   //Задание коэффициэнтов в ручном режиме

   "PID_Compact_Zone5".Retain.CtrlParams.Gain := "Param_PID".k_PID_Zona5.Gain; // Изменение коэф. П
   "PID_Compact_Zone5".Retain.CtrlParams.Ti := "Param_PID".k_PID_Zona5.I; // Изменение коэф И
   "PID_Compact_Zone5".Retain.CtrlParams.Td := "Param_PID".k_PID_Zona5.D; // Изменение коэф Д
END_REGION

REGION Network 11: ПИД - Зона 6
   // Выдержка
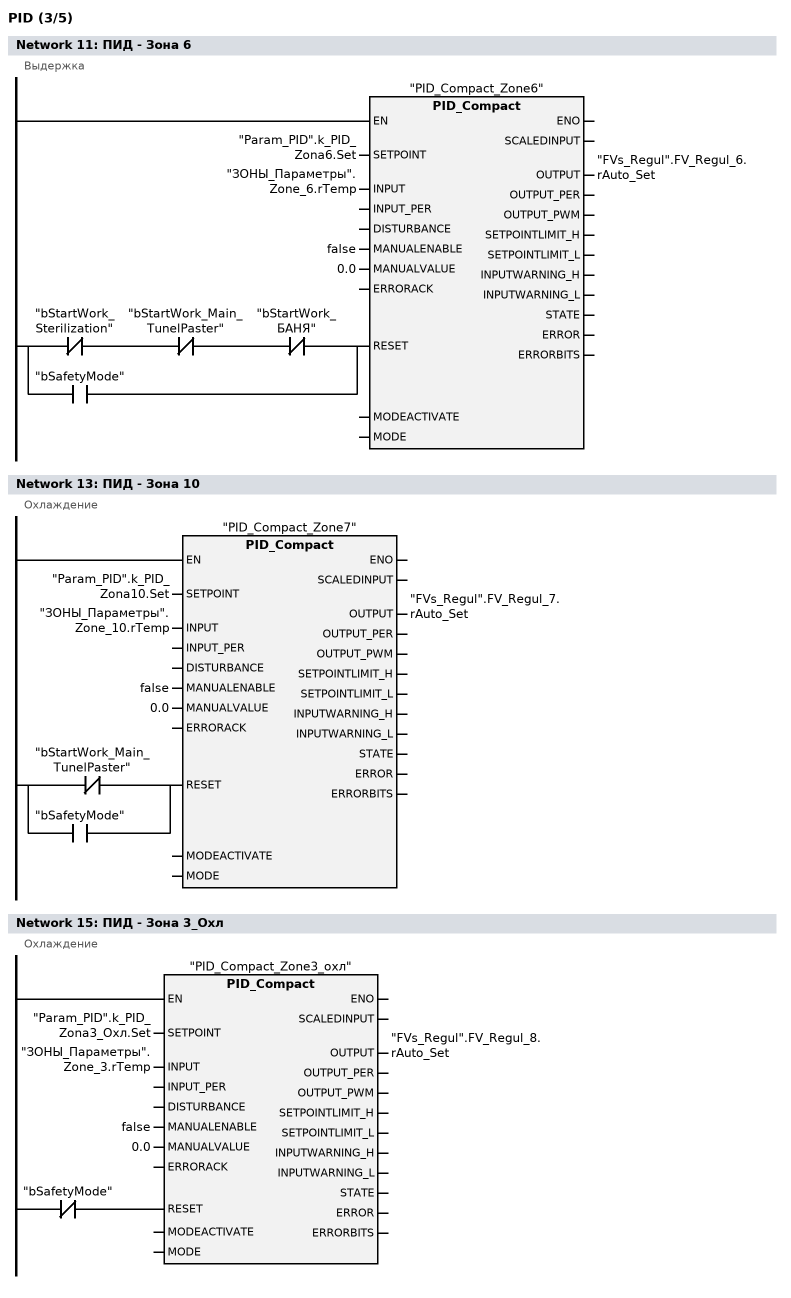
   "PID_Compact_Zone6"(Setpoint := "Param_PID".k_PID_Zona6.Set,   // PID_Compact
                       Input := "ЗОНЫ_Параметры".Zone_6.rTemp,
                       ManualEnable := false,
                       ManualValue := 0.0,
                       Reset := (NOT "bStartWork_Sterilization" AND NOT "bStartWork_Main_TunelPaster" AND NOT "bStartWork_БАНЯ") OR "bSafetyMode",
                       Output => "FVs_Regul".FV_Regul_6.rAuto_Set);
END_REGION

REGION Network 12 (SCL): Выбор типа ПИД Зона 6
   // 0 - Нагрев; 1 - Охлаждение
   //Режим работы ПИД - 0 - Нагрев; 1 - Охлаждение
   "PID_Compact_Zone6".Config.InvertControl := "bTypePID_Zone6";
   //Задание коэффициэнтов в ручном режиме

   "PID_Compact_Zone6".Retain.CtrlParams.Gain := "Param_PID".k_PID_Zona6.Gain; // Изменение коэф. П
   "PID_Compact_Zone6".Retain.CtrlParams.Ti := "Param_PID".k_PID_Zona6.I; // Изменение коэф И
   "PID_Compact_Zone6".Retain.CtrlParams.Td := "Param_PID".k_PID_Zona6.D; // Изменение коэф Д
END_REGION

REGION Network 13: ПИД - Зона 10
   // Охлаждение
   "PID_Compact_Zone7"(Setpoint := "Param_PID".k_PID_Zona10.Set,   // PID_Compact
                       Input := "ЗОНЫ_Параметры".Zone_10.rTemp,
                       ManualEnable := false,
                       ManualValue := 0.0,
                       Reset := NOT "bStartWork_Main_TunelPaster" OR "bSafetyMode",
                       Output => "FVs_Regul".FV_Regul_7.rAuto_Set);
END_REGION

REGION Network 14 (SCL): Выбор типа ПИД Зона 7
   // 0 - Нагрев; 1 - Охлаждение
   //Режим работы ПИД - 0 - Нагрев; 1 - Охлаждение
   "PID_Compact_Zone7".Config.InvertControl := TRUE;
   //Задание коэффициэнтов в ручном режиме

   "PID_Compact_Zone7".Retain.CtrlParams.Gain := "Param_PID".k_PID_Zona5_Охл.Gain; // Изменение коэф. П
   "PID_Compact_Zone7".Retain.CtrlParams.Ti := "Param_PID".k_PID_Zona5_Охл.I; // Изменение коэф И
   "PID_Compact_Zone7".Retain.CtrlParams.Td := "Param_PID".k_PID_Zona5_Охл.D; // Изменение коэф Д
END_REGION

REGION Network 15: ПИД - Зона 3_Охл
   // Охлаждение
   "PID_Compact_Zone3_охл"(Setpoint := "Param_PID".k_PID_Zona3_Охл.Set,   // PID_Compact
                           Input := "ЗОНЫ_Параметры".Zone_3.rTemp,
                           ManualEnable := false,
                           ManualValue := 0.0,
                           Reset := NOT "bSafetyMode",
                           Output => "FVs_Regul".FV_Regul_8.rAuto_Set);
END_REGION

REGION Network 16 (SCL): Выбор типа ПИД Зона 3_охл
   // 0 - Нагрев; 1 - Охлаждение
   //Режим работы ПИД - 0 - Нагрев; 1 - Охлаждение
   "PID_Compact_Zone3_охл".Config.InvertControl := TRUE;
   //Задание коэффициэнтов в ручном режиме

   "PID_Compact_Zone3_охл".Retain.CtrlParams.Gain := "Param_PID".k_PID_Zona3_Охл.Gain; // Изменение коэф. П
   "PID_Compact_Zone3_охл".Retain.CtrlParams.Ti := "Param_PID".k_PID_Zona3_Охл.I; // Изменение коэф И
   "PID_Compact_Zone3_охл".Retain.CtrlParams.Td := "Param_PID".k_PID_Zona3_Охл.D; // Изменение коэф Д
END_REGION

REGION Network 17: ПИД - Зона 4_Охл
   // Охлаждение
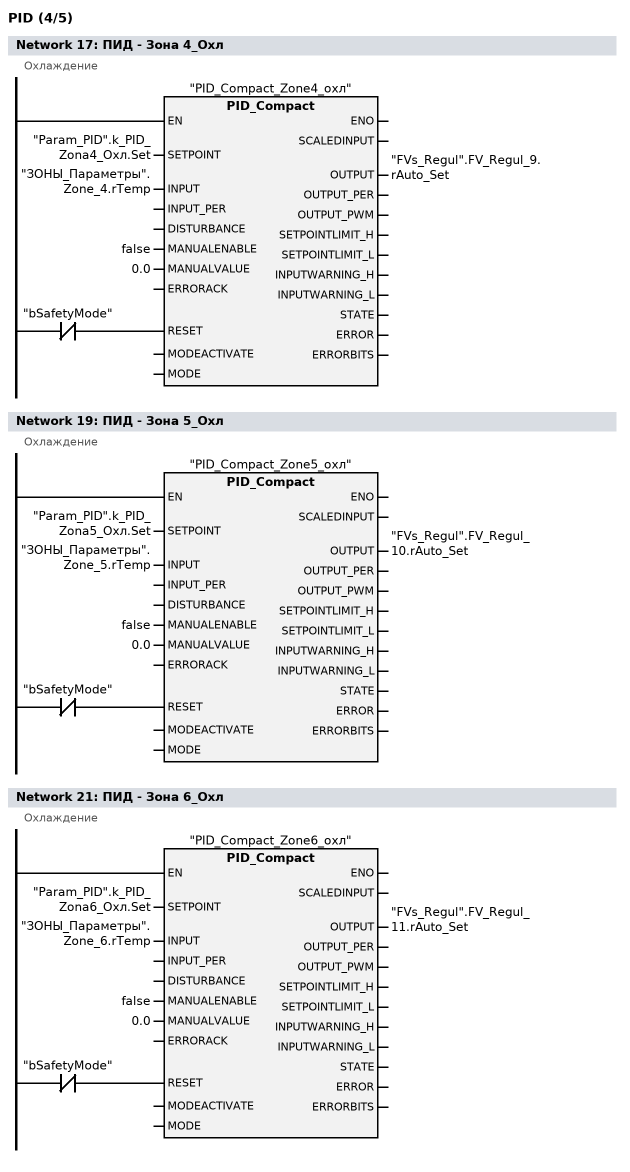
   "PID_Compact_Zone4_охл"(Setpoint := "Param_PID".k_PID_Zona4_Охл.Set,   // PID_Compact
                           Input := "ЗОНЫ_Параметры".Zone_4.rTemp,
                           ManualEnable := false,
                           ManualValue := 0.0,
                           Reset := NOT "bSafetyMode",
                           Output => "FVs_Regul".FV_Regul_9.rAuto_Set);
END_REGION

REGION Network 18 (SCL): Выбор типа ПИД Зона 4_охл
   // 0 - Нагрев; 1 - Охлаждение
   //Режим работы ПИД - 0 - Нагрев; 1 - Охлаждение
   "PID_Compact_Zone4_охл".Config.InvertControl := TRUE;
   //Задание коэффициэнтов в ручном режиме

   "PID_Compact_Zone4_охл".Retain.CtrlParams.Gain := "Param_PID".k_PID_Zona5_Охл.Gain; // Изменение коэф. П
   "PID_Compact_Zone4_охл".Retain.CtrlParams.Ti := "Param_PID".k_PID_Zona5_Охл.I; // Изменение коэф И
   "PID_Compact_Zone4_охл".Retain.CtrlParams.Td := "Param_PID".k_PID_Zona5_Охл.D; // Изменение коэф Д
END_REGION

REGION Network 19: ПИД - Зона 5_Охл
   // Охлаждение
   "PID_Compact_Zone5_охл"(Setpoint := "Param_PID".k_PID_Zona5_Охл.Set,   // PID_Compact
                           Input := "ЗОНЫ_Параметры".Zone_5.rTemp,
                           ManualEnable := false,
                           ManualValue := 0.0,
                           Reset := NOT "bSafetyMode",
                           Output => "FVs_Regul".FV_Regul_10.rAuto_Set);
END_REGION

REGION Network 20 (SCL): Выбор типа ПИД Зона 5_охл
   // 0 - Нагрев; 1 - Охлаждение
   //Режим работы ПИД - 0 - Нагрев; 1 - Охлаждение
   "PID_Compact_Zone5_охл".Config.InvertControl := TRUE;
   //Задание коэффициэнтов в ручном режиме

   "PID_Compact_Zone5_охл".Retain.CtrlParams.Gain := "Param_PID".k_PID_Zona5_Охл.Gain; // Изменение коэф. П
   "PID_Compact_Zone5_охл".Retain.CtrlParams.Ti := "Param_PID".k_PID_Zona5_Охл.I; // Изменение коэф И
   "PID_Compact_Zone5_охл".Retain.CtrlParams.Td := "Param_PID".k_PID_Zona5_Охл.D; // Изменение коэф Д
END_REGION

REGION Network 21: ПИД - Зона 6_Охл
   // Охлаждение
   "PID_Compact_Zone6_охл"(Setpoint := "Param_PID".k_PID_Zona6_Охл.Set,   // PID_Compact
                           Input := "ЗОНЫ_Параметры".Zone_6.rTemp,
                           ManualEnable := false,
                           ManualValue := 0.0,
                           Reset := NOT "bSafetyMode",
                           Output => "FVs_Regul".FV_Regul_11.rAuto_Set);
END_REGION

REGION Network 22 (SCL): Выбор типа ПИД Зона 6_охл
   // 0 - Нагрев; 1 - Охлаждение
   //Режим работы ПИД - 0 - Нагрев; 1 - Охлаждение
   "PID_Compact_Zone6_охл".Config.InvertControl := TRUE;
   //Задание коэффициэнтов в ручном режиме

   "PID_Compact_Zone6_охл".Retain.CtrlParams.Gain := "Param_PID".k_PID_Zona5_Охл.Gain; // Изменение коэф. П
   "PID_Compact_Zone6_охл".Retain.CtrlParams.Ti := "Param_PID".k_PID_Zona5_Охл.I; // Изменение коэф И
   "PID_Compact_Zone6_охл".Retain.CtrlParams.Td := "Param_PID".k_PID_Zona5_Охл.D; // Изменение коэф Д
END_REGION

REGION Network 23: ПИД - Зона 7_Охл
   // Охлаждение
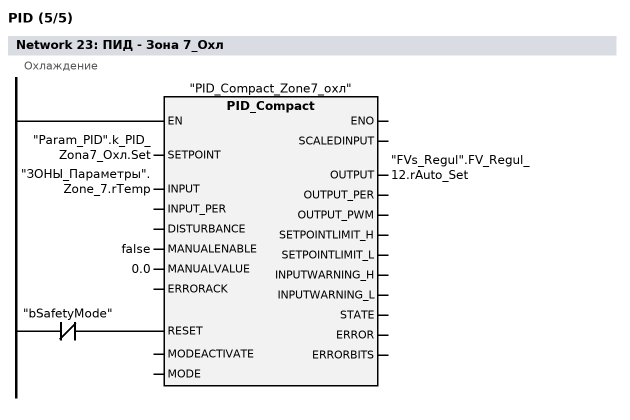
   "PID_Compact_Zone7_охл"(Setpoint := "Param_PID".k_PID_Zona7_Охл.Set,   // PID_Compact
                           Input := "ЗОНЫ_Параметры".Zone_7.rTemp,
                           ManualEnable := false,
                           ManualValue := 0.0,
                           Reset := NOT "bSafetyMode",
                           Output => "FVs_Regul".FV_Regul_12.rAuto_Set);
END_REGION

REGION Network 24 (SCL): Выбор типа ПИД Зона 7_охл
   // 0 - Нагрев; 1 - Охлаждение
   //Режим работы ПИД - 0 - Нагрев; 1 - Охлаждение
   "PID_Compact_Zone7_охл".Config.InvertControl := TRUE;
   //Задание коэффициэнтов в ручном режиме

   "PID_Compact_Zone7_охл".Retain.CtrlParams.Gain := "Param_PID".k_PID_Zona5_Охл.Gain; // Изменение коэф. П
   "PID_Compact_Zone7_охл".Retain.CtrlParams.Ti := "Param_PID".k_PID_Zona5_Охл.I; // Изменение коэф И
   "PID_Compact_Zone7_охл".Retain.CtrlParams.Td := "Param_PID".k_PID_Zona5_Охл.D; // Изменение коэф Д
END_REGION
END_ORGANIZATION_BLOCK

ORGANIZATION_BLOCK "Исполнительные устройств"   // OB123, LAD, ProgramCycle
TITLE = Работа физических устройств
{ S7_Optimized_Access := 'TRUE' }
VERSION : 0.1
// Насосы, клапана, и т.д.
   VAR_INPUT
      Initial_Call : Bool;   // Initial call of this OB
      Remanence : Bool;   // =True, if remanent data are available
   END_VAR
BEGIN

REGION Network 1: Аналогвые датчики
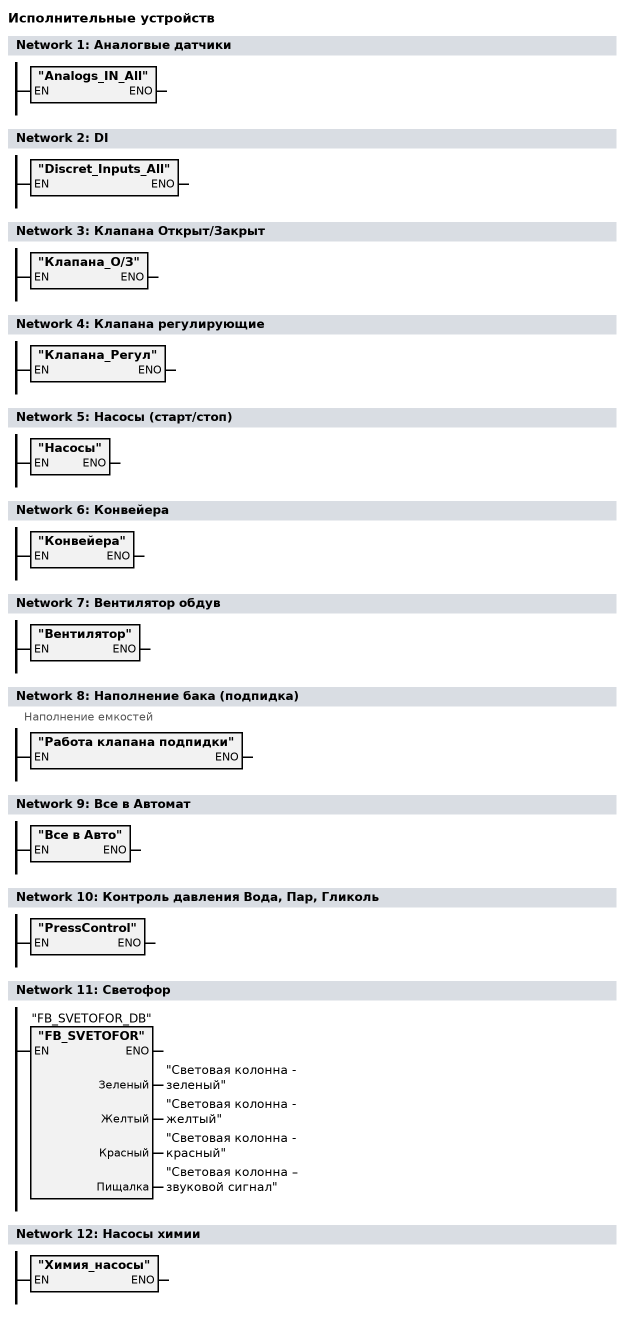
   RUNG wire#powerrail
      "Analogs_IN_All"()
   END_RUNG
   // the same network as SCL:
   "Analogs_IN_All"();
END_REGION

REGION Network 2: DI
   RUNG wire#powerrail
      "Discret_Inputs_All"()
   END_RUNG
   // the same network as SCL:
   "Discret_Inputs_All"();
END_REGION

REGION Network 3: Клапана Открыт/Закрыт
   RUNG wire#powerrail
      "Клапана_О/З"()
   END_RUNG
   // the same network as SCL:
   "Клапана_О/З"();
END_REGION

REGION Network 4: Клапана регулирующие
   RUNG wire#powerrail
      "Клапана_Регул"()
   END_RUNG
   // the same network as SCL:
   "Клапана_Регул"();
END_REGION

REGION Network 5: Насосы (старт/стоп)
   RUNG wire#powerrail
      "Насосы"()
   END_RUNG
   // the same network as SCL:
   "Насосы"();
END_REGION

REGION Network 6: Конвейера
   RUNG wire#powerrail
      "Конвейера"()
   END_RUNG
   // the same network as SCL:
   "Конвейера"();
END_REGION

REGION Network 7: Вентилятор обдув
   RUNG wire#powerrail
      "Вентилятор"()
   END_RUNG
   // the same network as SCL:
   "Вентилятор"();
END_REGION

REGION Network 8: Наполнение бака (подпидка)
   // Наполнение емкостей
   RUNG wire#powerrail
      "Работа клапана подпидки"()
   END_RUNG
   // the same network as SCL:
   "Работа клапана подпидки"();
END_REGION

REGION Network 9: Все в Автомат
   RUNG wire#powerrail
      "Все в Авто"()
   END_RUNG
   // the same network as SCL:
   "Все в Авто"();
END_REGION

REGION Network 10: Контроль давления Вода, Пар, Гликоль
   RUNG wire#powerrail
      "PressControl"()
   END_RUNG
   // the same network as SCL:
   "PressControl"();
END_REGION

REGION Network 11: Светофор
   RUNG wire#powerrail
      "FB_SVETOFOR_DB"(Зеленый => "Световая колонна - зеленый", Желтый => "Световая колонна - желтый", Красный => "Световая колонна - красный", Пищалка => "Световая колонна – звуковой сигнал")
   END_RUNG
   // the same network as SCL:
   "FB_SVETOFOR_DB"(Зеленый => "Световая колонна - зеленый",   // "FB_SVETOFOR"
                    Желтый => "Световая колонна - желтый",
                    Красный => "Световая колонна - красный",
                    Пищалка => "Световая колонна – звуковой сигнал");
END_REGION

REGION Network 12: Насосы химии
   RUNG wire#powerrail
      "Химия_насосы"()
   END_RUNG
   // the same network as SCL:
   "Химия_насосы"();
END_REGION
END_ORGANIZATION_BLOCK

ORGANIZATION_BLOCK "Пастеризация"   // OB124, LAD, ProgramCycle
TITLE = "Main Program Sweep (Cycle)"
{ S7_Optimized_Access := 'TRUE' }
VERSION : 0.1
   VAR_INPUT
      Initial_Call : Bool;   // Initial call of this OB
      Remanence : Bool;   // =True, if remanent data are available
   END_VAR
BEGIN

REGION Network 1: Старт Пастеризация
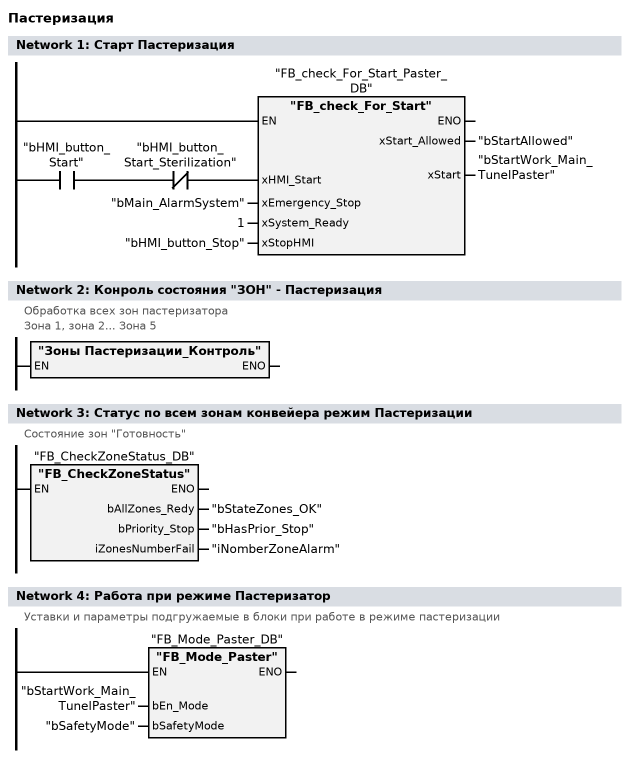
   RUNG wire#powerrail
      "FB_check_For_Start_Paster_DB"(xHMI_Start := wire#w1, xEmergency_Stop := "bMain_AlarmSystem", xSystem_Ready := 1, xStopHMI := "bHMI_button_Stop", xStart_Allowed => "bStartAllowed", xStart => "bStartWork_Main_TunelPaster")
   END_RUNG
   RUNG wire#powerrail
      Contact( "bHMI_button_Start" )
      I_Contact( "bHMI_button_Start_Sterilization" )
   END_RUNG wire#w1
   // the same network as SCL:
   "FB_check_For_Start_Paster_DB"(xHMI_Start := "bHMI_button_Start" AND NOT "bHMI_button_Start_Sterilization",   // "FB_check_For_Start"
                           xEmergency_Stop := "bMain_AlarmSystem",
                           xSystem_Ready := 1,
                           xStopHMI := "bHMI_button_Stop",
                           xStart_Allowed => "bStartAllowed",
                           xStart => "bStartWork_Main_TunelPaster");
END_REGION

REGION Network 2: Конроль состояния "ЗОН" - Пастеризация
   // Обработка всех зон пастеризатора
   // Зона 1, зона 2... Зона 5
   RUNG wire#powerrail
      "Зоны Пастеризации_Контроль"()
   END_RUNG
   // the same network as SCL:
   "Зоны Пастеризации_Контроль"();
END_REGION

REGION Network 3: Статус по всем зонам конвейера режим Пастеризации
   // Состояние зон "Готовность"
   RUNG wire#powerrail
      "FB_CheckZoneStatus_DB"(bAllZones_Redy => "bStateZones_OK", bPriority_Stop => "bHasPrior_Stop", iZonesNumberFail => "iNomberZoneAlarm")
   END_RUNG
   // the same network as SCL:
   "FB_CheckZoneStatus_DB"(bAllZones_Redy => "bStateZones_OK",   // "FB_CheckZoneStatus"
                           bPriority_Stop => "bHasPrior_Stop",
                           iZonesNumberFail => "iNomberZoneAlarm");
END_REGION

REGION Network 4: Работа при режиме Пастеризатор
   // Уставки и параметры подгружаемые в блоки при работе в режиме пастеризации
   RUNG wire#powerrail
      "FB_Mode_Paster_DB"(bEn_Mode := "bStartWork_Main_TunelPaster", bSafetyMode := "bSafetyMode")
   END_RUNG
   // the same network as SCL:
   "FB_Mode_Paster_DB"(bEn_Mode := "bStartWork_Main_TunelPaster", bSafetyMode := "bSafetyMode");   // "FB_Mode_Paster"
END_REGION
END_ORGANIZATION_BLOCK

ORGANIZATION_BLOCK "Баня"   // OB125, LAD, ProgramCycle
TITLE = "Main Program Sweep (Cycle)"
{ S7_Optimized_Access := 'TRUE' }
VERSION : 0.1
   VAR_INPUT
      Initial_Call : Bool;   // Initial call of this OB
      Remanence : Bool;   // =True, if remanent data are available
   END_VAR
BEGIN

REGION Network 1: Старт БАНЯ
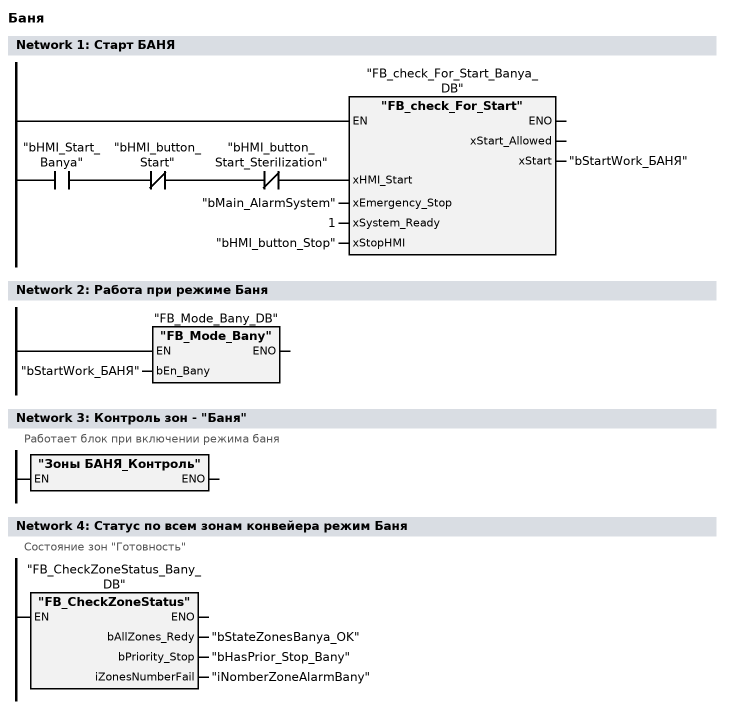
   RUNG wire#powerrail
      "FB_check_For_Start_Banya_DB"(xHMI_Start := wire#w1, xEmergency_Stop := "bMain_AlarmSystem", xSystem_Ready := 1, xStopHMI := "bHMI_button_Stop", xStart_Allowed =>, xStart => "bStartWork_БАНЯ")
   END_RUNG
   RUNG wire#powerrail
      Contact( "bHMI_Start_Banya" )
      I_Contact( "bHMI_button_Start" )
      I_Contact( "bHMI_button_Start_Sterilization" )
   END_RUNG wire#w1
   // the same network as SCL:
   "FB_check_For_Start_Banya_DB"(xHMI_Start := "bHMI_Start_Banya" AND NOT "bHMI_button_Start" AND NOT "bHMI_button_Start_Sterilization",   // "FB_check_For_Start"
                           xEmergency_Stop := "bMain_AlarmSystem",
                           xSystem_Ready := 1,
                           xStopHMI := "bHMI_button_Stop",
                           xStart => "bStartWork_БАНЯ");
END_REGION

REGION Network 2: Работа при режиме Баня
   RUNG wire#powerrail
      "FB_Mode_Bany_DB"(bEn_Bany := "bStartWork_БАНЯ")
   END_RUNG
   // the same network as SCL:
   "FB_Mode_Bany_DB"(bEn_Bany := "bStartWork_БАНЯ");   // "FB_Mode_Bany"
END_REGION

REGION Network 3: Контроль зон - "Баня"
   // Работает блок при включении режима баня
   RUNG wire#powerrail
      "Зоны БАНЯ_Контроль"()
   END_RUNG
   // the same network as SCL:
   "Зоны БАНЯ_Контроль"();
END_REGION

REGION Network 4: Статус по всем зонам конвейера режим Баня
   // Состояние зон "Готовность"
   RUNG wire#powerrail
      "FB_CheckZoneStatus_Bany_DB"(bAllZones_Redy => "bStateZonesBanya_OK", bPriority_Stop => "bHasPrior_Stop_Bany", iZonesNumberFail => "iNomberZoneAlarmBany")
   END_RUNG
   // the same network as SCL:
   "FB_CheckZoneStatus_Bany_DB"(bAllZones_Redy => "bStateZonesBanya_OK",   // "FB_CheckZoneStatus"
                           bPriority_Stop => "bHasPrior_Stop_Bany",
                           iZonesNumberFail => "iNomberZoneAlarmBany");
END_REGION
END_ORGANIZATION_BLOCK

ORGANIZATION_BLOCK "Стирилизация"   // OB126, LAD, ProgramCycle
TITLE = "Main Program Sweep (Cycle)"
{ S7_Optimized_Access := 'TRUE' }
VERSION : 0.1
   VAR_INPUT
      Initial_Call : Bool;   // Initial call of this OB
      Remanence : Bool;   // =True, if remanent data are available
   END_VAR
BEGIN

REGION Network 2: Старт и проверка старта "Стерилизации"
   // Проверка на разрешение старта режима "Стерилизация"
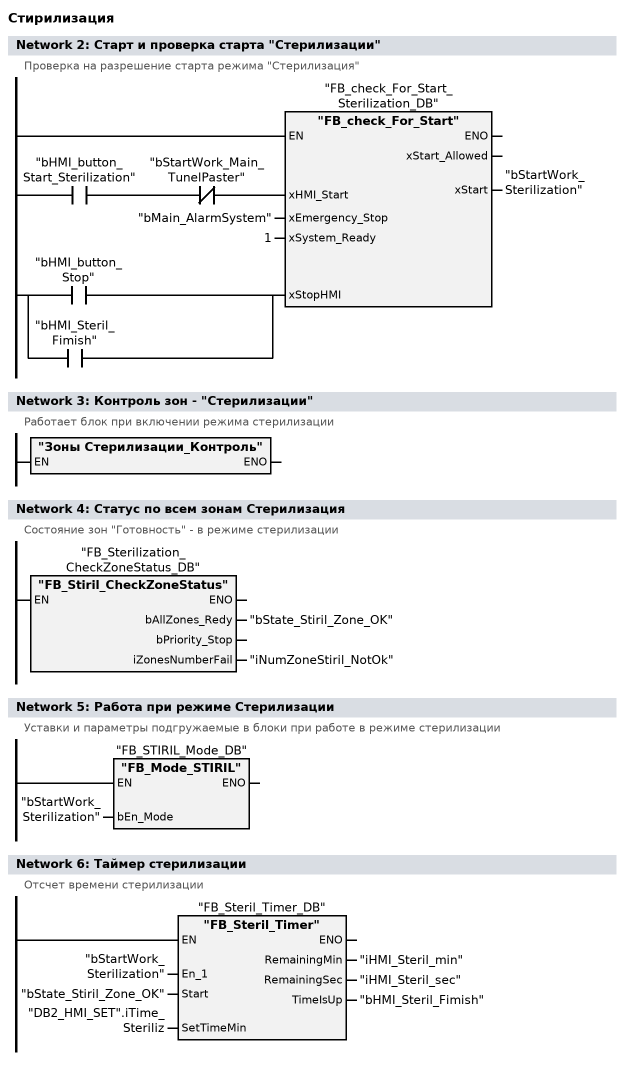
   RUNG wire#powerrail
      "FB_check_For_Start_Sterilization_DB"(xHMI_Start := wire#w1, xStopHMI := wire#w2, xEmergency_Stop := "bMain_AlarmSystem", xSystem_Ready := 1, xStart_Allowed =>, xStart => "bStartWork_Sterilization")
   END_RUNG
   RUNG wire#powerrail
      Contact( "bHMI_button_Start_Sterilization" )
      I_Contact( "bStartWork_Main_TunelPaster" )
   END_RUNG wire#w1
   RUNG wire#powerrail
      Contact( "bHMI_button_Stop" )
   END_RUNG wire#w2
   RUNG wire#powerrail
      Contact( "bHMI_Steril_Fimish" )
   END_RUNG wire#w2
   // the same network as SCL:
   "FB_check_For_Start_Sterilization_DB"(xHMI_Start := "bHMI_button_Start_Sterilization" AND NOT "bStartWork_Main_TunelPaster",   // "FB_check_For_Start"
                           xEmergency_Stop := "bMain_AlarmSystem",
                           xSystem_Ready := 1,
                           xStopHMI := "bHMI_button_Stop" OR "bHMI_Steril_Fimish",
                           xStart => "bStartWork_Sterilization");
END_REGION

REGION Network 3: Контроль зон - "Стерилизации"
   // Работает блок при включении режима стерилизации
   RUNG wire#powerrail
      "Зоны Стерилизации_Контроль"()
   END_RUNG
   // the same network as SCL:
   "Зоны Стерилизации_Контроль"();
END_REGION

REGION Network 4: Статус по всем зонам Стерилизация
   // Состояние зон "Готовность" - в режиме стерилизации
   RUNG wire#powerrail
      "FB_Sterilization_CheckZoneStatus_DB"(bAllZones_Redy => "bState_Stiril_Zone_OK", bPriority_Stop =>, iZonesNumberFail => "iNumZoneStiril_NotOk")
   END_RUNG
   // the same network as SCL:
   "FB_Sterilization_CheckZoneStatus_DB"(bAllZones_Redy => "bState_Stiril_Zone_OK",   // "FB_Stiril_CheckZoneStatus"
                           iZonesNumberFail => "iNumZoneStiril_NotOk");
END_REGION

REGION Network 5: Работа при режиме Стерилизации
   // Уставки и параметры подгружаемые в блоки при работе в режиме стерилизации
   RUNG wire#powerrail
      "FB_STIRIL_Mode_DB"(bEn_Mode := "bStartWork_Sterilization")
   END_RUNG
   // the same network as SCL:
   "FB_STIRIL_Mode_DB"(bEn_Mode := "bStartWork_Sterilization");   // "FB_Mode_STIRIL"
END_REGION

REGION Network 6: Таймер стерилизации
   // Отсчет времени стерилизации
   RUNG wire#powerrail
      "FB_Steril_Timer_DB"(En_1 := "bStartWork_Sterilization", Start := "bState_Stiril_Zone_OK", SetTimeMin := "DB2_HMI_SET".iTime_Steriliz, RemainingMin => "iHMI_Steril_min", RemainingSec => "iHMI_Steril_sec", TimeIsUp => "bHMI_Steril_Fimish")
   END_RUNG
   // the same network as SCL:
   "FB_Steril_Timer_DB"(En_1 := "bStartWork_Sterilization",   // "FB_Steril_Timer"
                        Start := "bState_Stiril_Zone_OK",
                        SetTimeMin := "DB2_HMI_SET".iTime_Steriliz,
                        RemainingMin => "iHMI_Steril_min",
                        RemainingSec => "iHMI_Steril_sec",
                        TimeIsUp => "bHMI_Steril_Fimish");
END_REGION

REGION Network 7 (SCL): Окно окончания стирилизации
   IF "bHMI_Steril_Fimish" THEN
       "iHMIWind_FinishStiril" := 148;
   END_IF;
END_REGION
END_ORGANIZATION_BLOCK

ORGANIZATION_BLOCK "RS_485"   // OB127, LAD, ProgramCycle
TITLE = "Main Program Sweep (Cycle)"
{ S7_Optimized_Access := 'TRUE' }
VERSION : 0.1
   VAR_INPUT
      Initial_Call : Bool;   // Initial call of this OB
      Remanence : Bool;   // =True, if remanent data are available
   END_VAR
   VAR_TEMP
      Test_Out : Int;
      Test_reaL : Real;
      Test_Real_Out : Real;
      off : Bool;
   END_VAR
BEGIN

REGION Network 1: Счетчик для RS485
   // Для последовательной обработки запросов по RS485
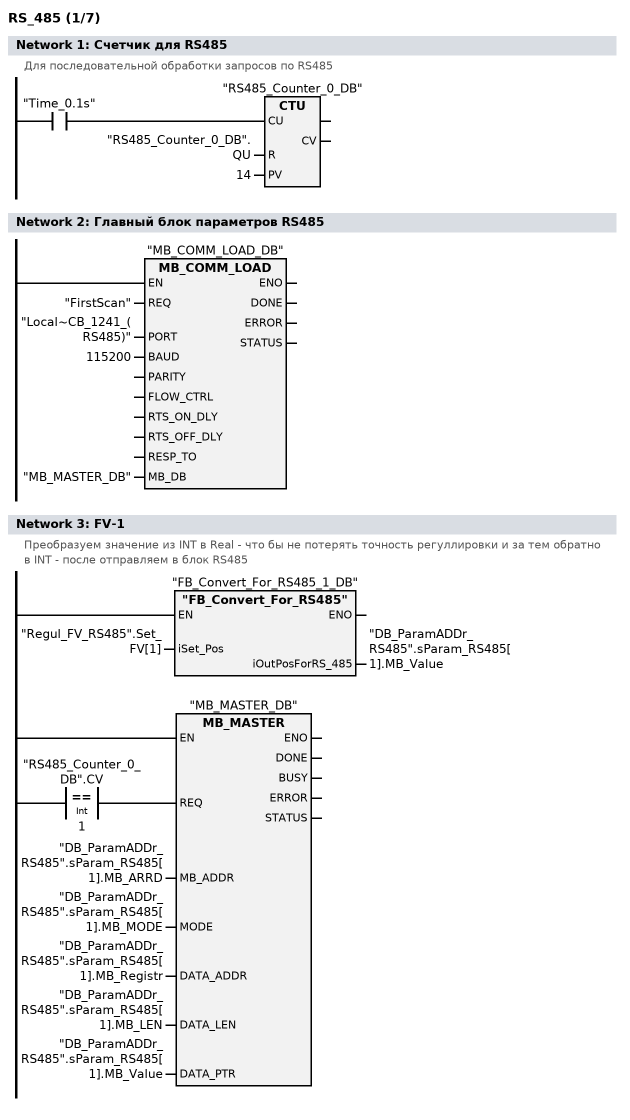
   "RS485_Counter_0_DB".CTU(CU := "Time_0.1s", R := "RS485_Counter_0_DB".QU, PV := 14);
END_REGION

REGION Network 2: Главный блок параметров RS485
   "MB_COMM_LOAD_DB"(REQ := "FirstScan",   // MB_COMM_LOAD
                     PORT := "Local~CB_1241_(RS485)",
                     BAUD := 115200,
                     MB_DB := "MB_MASTER_DB");
END_REGION

REGION Network 3: FV-1
   // Преобразуем значение из INT в Real - что бы не потерять точность регуллировки и за тем обратно в INT - после отправляем в блок RS485
   "FB_Convert_For_RS485_1_DB"(iSet_Pos := "Regul_FV_RS485".Set_FV[1],   // "FB_Convert_For_RS485"
                           iOutPosForRS_485 => "DB_ParamADDr_RS485".sParam_RS485[1].MB_Value);
   "MB_MASTER_DB"(REQ := "RS485_Counter_0_DB".CV = 1,   // MB_MASTER
                  MB_ADDR := "DB_ParamADDr_RS485".sParam_RS485[1].MB_ARRD,
                  MODE := "DB_ParamADDr_RS485".sParam_RS485[1].MB_MODE,
                  DATA_ADDR := "DB_ParamADDr_RS485".sParam_RS485[1].MB_Registr,
                  DATA_LEN := "DB_ParamADDr_RS485".sParam_RS485[1].MB_LEN,
                  DATA_PTR := "DB_ParamADDr_RS485".sParam_RS485[1].MB_Value);
END_REGION

REGION Network 4: FV-2
   // Преобразуем значение из INT в Real - что бы не потерять точность регуллировки и за тем обратно в INT - после отправляем в блок RS485
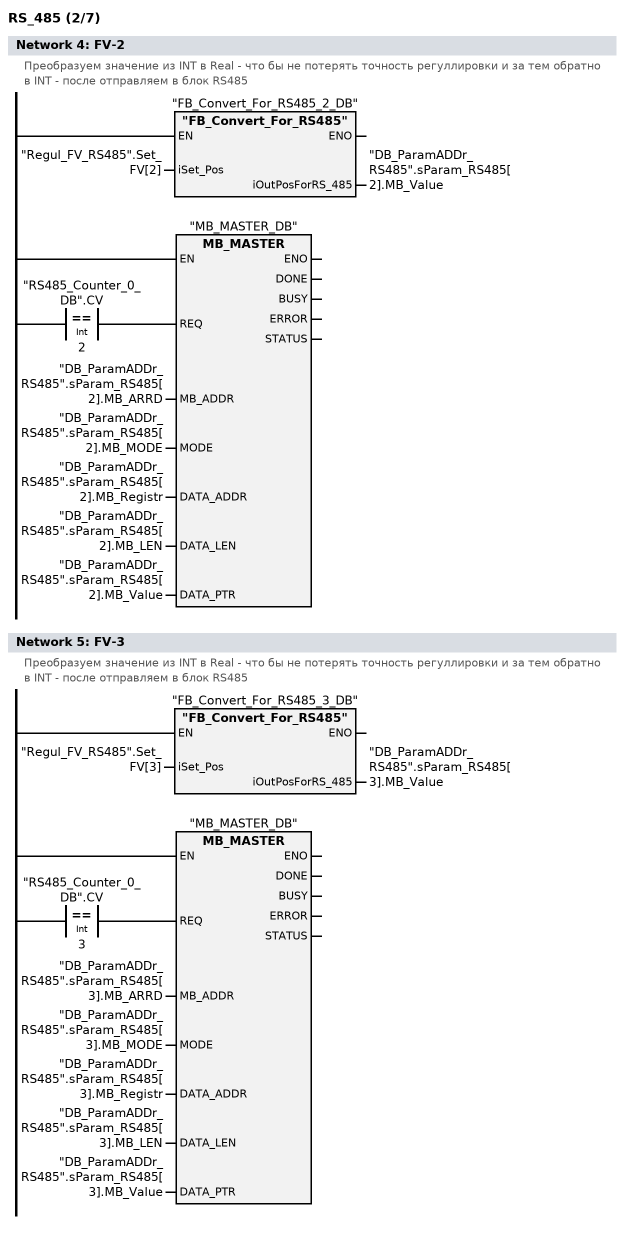
   "FB_Convert_For_RS485_2_DB"(iSet_Pos := "Regul_FV_RS485".Set_FV[2],   // "FB_Convert_For_RS485"
                           iOutPosForRS_485 => "DB_ParamADDr_RS485".sParam_RS485[2].MB_Value);
   "MB_MASTER_DB"(REQ := "RS485_Counter_0_DB".CV = 2,   // MB_MASTER
                  MB_ADDR := "DB_ParamADDr_RS485".sParam_RS485[2].MB_ARRD,
                  MODE := "DB_ParamADDr_RS485".sParam_RS485[2].MB_MODE,
                  DATA_ADDR := "DB_ParamADDr_RS485".sParam_RS485[2].MB_Registr,
                  DATA_LEN := "DB_ParamADDr_RS485".sParam_RS485[2].MB_LEN,
                  DATA_PTR := "DB_ParamADDr_RS485".sParam_RS485[2].MB_Value);
END_REGION

REGION Network 5: FV-3
   // Преобразуем значение из INT в Real - что бы не потерять точность регуллировки и за тем обратно в INT - после отправляем в блок RS485
   "FB_Convert_For_RS485_3_DB"(iSet_Pos := "Regul_FV_RS485".Set_FV[3],   // "FB_Convert_For_RS485"
                           iOutPosForRS_485 => "DB_ParamADDr_RS485".sParam_RS485[3].MB_Value);
   "MB_MASTER_DB"(REQ := "RS485_Counter_0_DB".CV = 3,   // MB_MASTER
                  MB_ADDR := "DB_ParamADDr_RS485".sParam_RS485[3].MB_ARRD,
                  MODE := "DB_ParamADDr_RS485".sParam_RS485[3].MB_MODE,
                  DATA_ADDR := "DB_ParamADDr_RS485".sParam_RS485[3].MB_Registr,
                  DATA_LEN := "DB_ParamADDr_RS485".sParam_RS485[3].MB_LEN,
                  DATA_PTR := "DB_ParamADDr_RS485".sParam_RS485[3].MB_Value);
END_REGION

REGION Network 6: FV-4
   // Преобразуем значение из INT в Real - что бы не потерять точность регуллировки и за тем обратно в INT - после отправляем в блок RS485
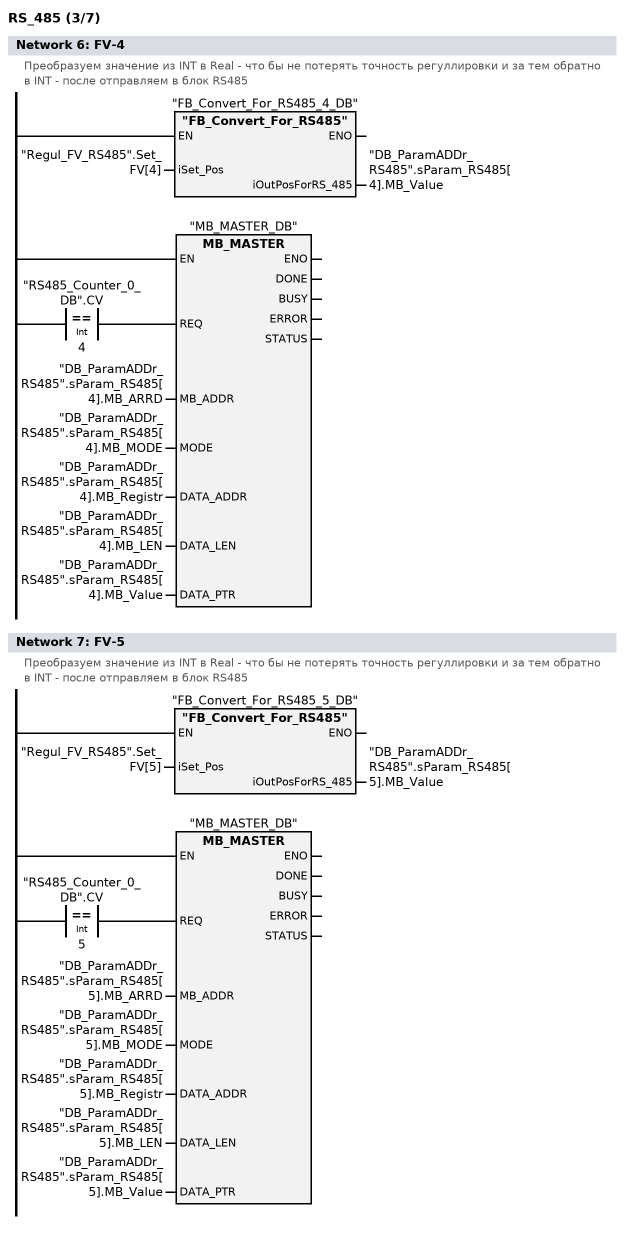
   "FB_Convert_For_RS485_4_DB"(iSet_Pos := "Regul_FV_RS485".Set_FV[4],   // "FB_Convert_For_RS485"
                           iOutPosForRS_485 => "DB_ParamADDr_RS485".sParam_RS485[4].MB_Value);
   "MB_MASTER_DB"(REQ := "RS485_Counter_0_DB".CV = 4,   // MB_MASTER
                  MB_ADDR := "DB_ParamADDr_RS485".sParam_RS485[4].MB_ARRD,
                  MODE := "DB_ParamADDr_RS485".sParam_RS485[4].MB_MODE,
                  DATA_ADDR := "DB_ParamADDr_RS485".sParam_RS485[4].MB_Registr,
                  DATA_LEN := "DB_ParamADDr_RS485".sParam_RS485[4].MB_LEN,
                  DATA_PTR := "DB_ParamADDr_RS485".sParam_RS485[4].MB_Value);
END_REGION

REGION Network 7: FV-5
   // Преобразуем значение из INT в Real - что бы не потерять точность регуллировки и за тем обратно в INT - после отправляем в блок RS485
   "FB_Convert_For_RS485_5_DB"(iSet_Pos := "Regul_FV_RS485".Set_FV[5],   // "FB_Convert_For_RS485"
                           iOutPosForRS_485 => "DB_ParamADDr_RS485".sParam_RS485[5].MB_Value);
   "MB_MASTER_DB"(REQ := "RS485_Counter_0_DB".CV = 5,   // MB_MASTER
                  MB_ADDR := "DB_ParamADDr_RS485".sParam_RS485[5].MB_ARRD,
                  MODE := "DB_ParamADDr_RS485".sParam_RS485[5].MB_MODE,
                  DATA_ADDR := "DB_ParamADDr_RS485".sParam_RS485[5].MB_Registr,
                  DATA_LEN := "DB_ParamADDr_RS485".sParam_RS485[5].MB_LEN,
                  DATA_PTR := "DB_ParamADDr_RS485".sParam_RS485[5].MB_Value);
END_REGION

REGION Network 8: FV-6
   // Преобразуем значение из INT в Real - что бы не потерять точность регуллировки и за тем обратно в INT - после отправляем в блок RS485
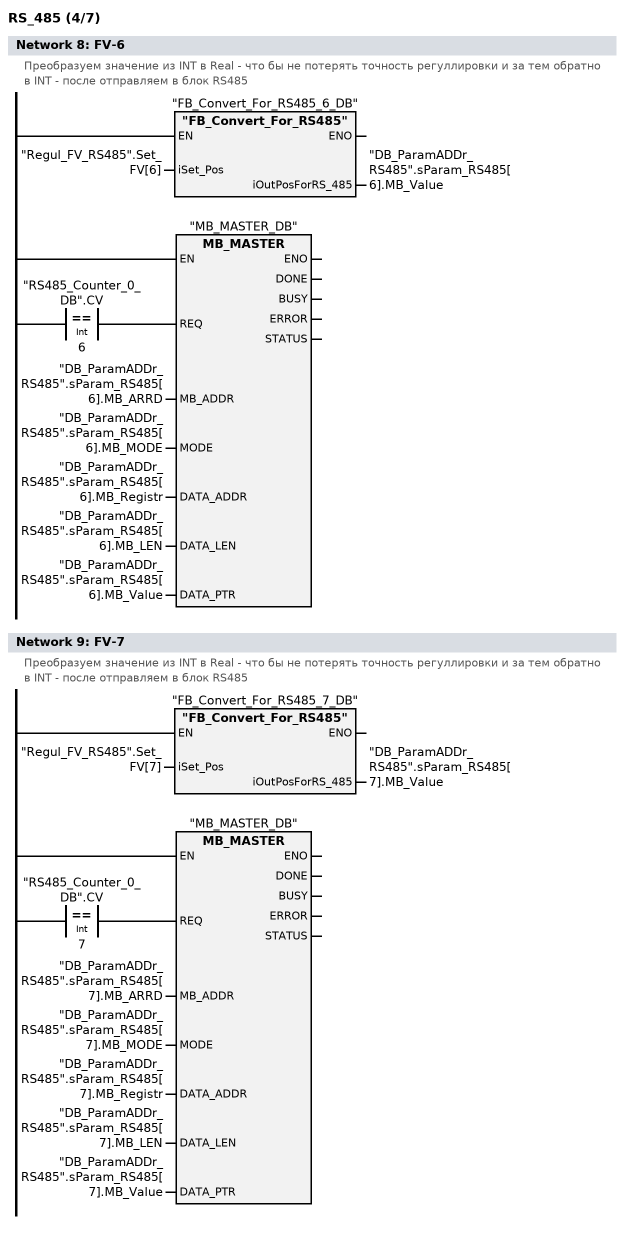
   "FB_Convert_For_RS485_6_DB"(iSet_Pos := "Regul_FV_RS485".Set_FV[6],   // "FB_Convert_For_RS485"
                           iOutPosForRS_485 => "DB_ParamADDr_RS485".sParam_RS485[6].MB_Value);
   "MB_MASTER_DB"(REQ := "RS485_Counter_0_DB".CV = 6,   // MB_MASTER
                  MB_ADDR := "DB_ParamADDr_RS485".sParam_RS485[6].MB_ARRD,
                  MODE := "DB_ParamADDr_RS485".sParam_RS485[6].MB_MODE,
                  DATA_ADDR := "DB_ParamADDr_RS485".sParam_RS485[6].MB_Registr,
                  DATA_LEN := "DB_ParamADDr_RS485".sParam_RS485[6].MB_LEN,
                  DATA_PTR := "DB_ParamADDr_RS485".sParam_RS485[6].MB_Value);
END_REGION

REGION Network 9: FV-7
   // Преобразуем значение из INT в Real - что бы не потерять точность регуллировки и за тем обратно в INT - после отправляем в блок RS485
   "FB_Convert_For_RS485_7_DB"(iSet_Pos := "Regul_FV_RS485".Set_FV[7],   // "FB_Convert_For_RS485"
                           iOutPosForRS_485 => "DB_ParamADDr_RS485".sParam_RS485[7].MB_Value);
   "MB_MASTER_DB"(REQ := "RS485_Counter_0_DB".CV = 7,   // MB_MASTER
                  MB_ADDR := "DB_ParamADDr_RS485".sParam_RS485[7].MB_ARRD,
                  MODE := "DB_ParamADDr_RS485".sParam_RS485[7].MB_MODE,
                  DATA_ADDR := "DB_ParamADDr_RS485".sParam_RS485[7].MB_Registr,
                  DATA_LEN := "DB_ParamADDr_RS485".sParam_RS485[7].MB_LEN,
                  DATA_PTR := "DB_ParamADDr_RS485".sParam_RS485[7].MB_Value);
END_REGION

REGION Network 10: FV-8
   // Преобразуем значение из INT в Real - что бы не потерять точность регуллировки и за тем обратно в INT - после отправляем в блок RS485
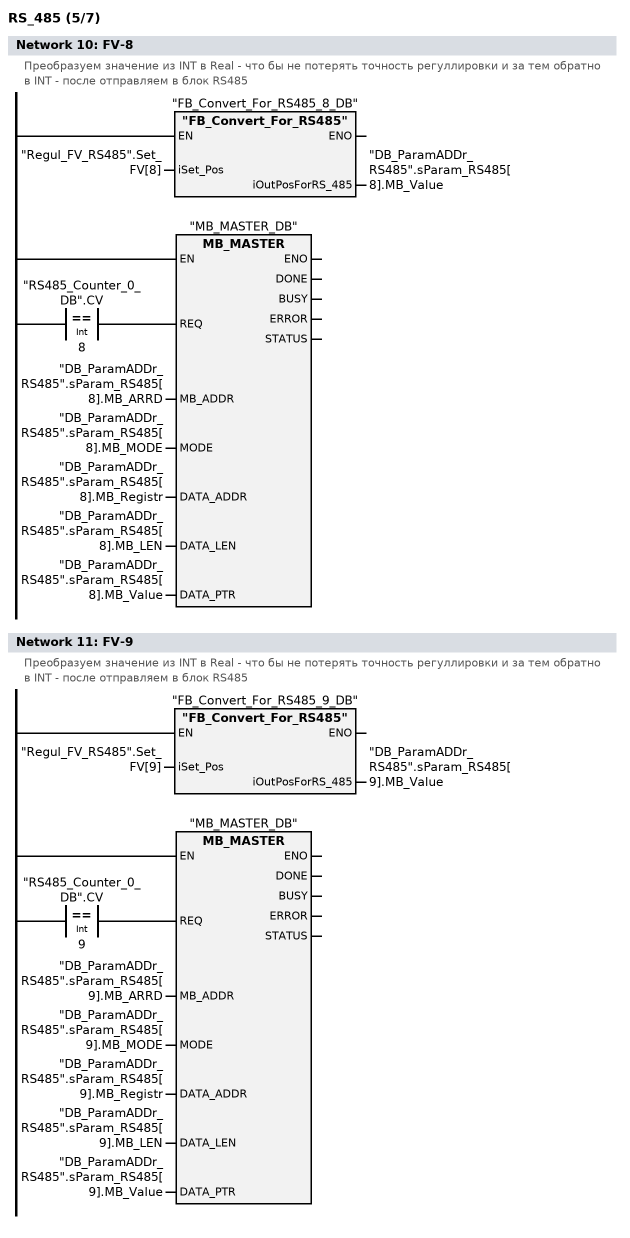
   "FB_Convert_For_RS485_8_DB"(iSet_Pos := "Regul_FV_RS485".Set_FV[8],   // "FB_Convert_For_RS485"
                           iOutPosForRS_485 => "DB_ParamADDr_RS485".sParam_RS485[8].MB_Value);
   "MB_MASTER_DB"(REQ := "RS485_Counter_0_DB".CV = 8,   // MB_MASTER
                  MB_ADDR := "DB_ParamADDr_RS485".sParam_RS485[8].MB_ARRD,
                  MODE := "DB_ParamADDr_RS485".sParam_RS485[8].MB_MODE,
                  DATA_ADDR := "DB_ParamADDr_RS485".sParam_RS485[8].MB_Registr,
                  DATA_LEN := "DB_ParamADDr_RS485".sParam_RS485[8].MB_LEN,
                  DATA_PTR := "DB_ParamADDr_RS485".sParam_RS485[8].MB_Value);
END_REGION

REGION Network 11: FV-9
   // Преобразуем значение из INT в Real - что бы не потерять точность регуллировки и за тем обратно в INT - после отправляем в блок RS485
   "FB_Convert_For_RS485_9_DB"(iSet_Pos := "Regul_FV_RS485".Set_FV[9],   // "FB_Convert_For_RS485"
                           iOutPosForRS_485 => "DB_ParamADDr_RS485".sParam_RS485[9].MB_Value);
   "MB_MASTER_DB"(REQ := "RS485_Counter_0_DB".CV = 9,   // MB_MASTER
                  MB_ADDR := "DB_ParamADDr_RS485".sParam_RS485[9].MB_ARRD,
                  MODE := "DB_ParamADDr_RS485".sParam_RS485[9].MB_MODE,
                  DATA_ADDR := "DB_ParamADDr_RS485".sParam_RS485[9].MB_Registr,
                  DATA_LEN := "DB_ParamADDr_RS485".sParam_RS485[9].MB_LEN,
                  DATA_PTR := "DB_ParamADDr_RS485".sParam_RS485[9].MB_Value);
END_REGION

REGION Network 12: FV-10
   // Преобразуем значение из INT в Real - что бы не потерять точность регуллировки и за тем обратно в INT - после отправляем в блок RS485
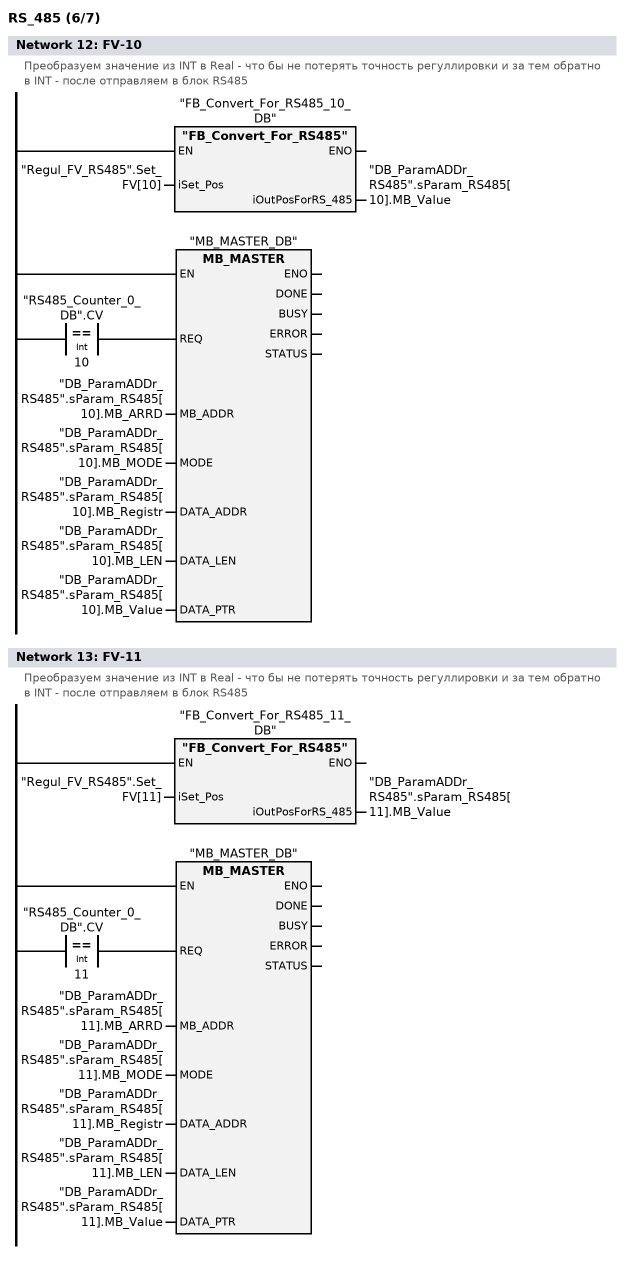
   "FB_Convert_For_RS485_10_DB"(iSet_Pos := "Regul_FV_RS485".Set_FV[10],   // "FB_Convert_For_RS485"
                           iOutPosForRS_485 => "DB_ParamADDr_RS485".sParam_RS485[10].MB_Value);
   "MB_MASTER_DB"(REQ := "RS485_Counter_0_DB".CV = 10,   // MB_MASTER
                  MB_ADDR := "DB_ParamADDr_RS485".sParam_RS485[10].MB_ARRD,
                  MODE := "DB_ParamADDr_RS485".sParam_RS485[10].MB_MODE,
                  DATA_ADDR := "DB_ParamADDr_RS485".sParam_RS485[10].MB_Registr,
                  DATA_LEN := "DB_ParamADDr_RS485".sParam_RS485[10].MB_LEN,
                  DATA_PTR := "DB_ParamADDr_RS485".sParam_RS485[10].MB_Value);
END_REGION

REGION Network 13: FV-11
   // Преобразуем значение из INT в Real - что бы не потерять точность регуллировки и за тем обратно в INT - после отправляем в блок RS485
   "FB_Convert_For_RS485_11_DB"(iSet_Pos := "Regul_FV_RS485".Set_FV[11],   // "FB_Convert_For_RS485"
                           iOutPosForRS_485 => "DB_ParamADDr_RS485".sParam_RS485[11].MB_Value);
   "MB_MASTER_DB"(REQ := "RS485_Counter_0_DB".CV = 11,   // MB_MASTER
                  MB_ADDR := "DB_ParamADDr_RS485".sParam_RS485[11].MB_ARRD,
                  MODE := "DB_ParamADDr_RS485".sParam_RS485[11].MB_MODE,
                  DATA_ADDR := "DB_ParamADDr_RS485".sParam_RS485[11].MB_Registr,
                  DATA_LEN := "DB_ParamADDr_RS485".sParam_RS485[11].MB_LEN,
                  DATA_PTR := "DB_ParamADDr_RS485".sParam_RS485[11].MB_Value);
END_REGION

REGION Network 14: FV-12
   // Преобразуем значение из INT в Real - что бы не потерять точность регуллировки и за тем обратно в INT - после отправляем в блок RS485
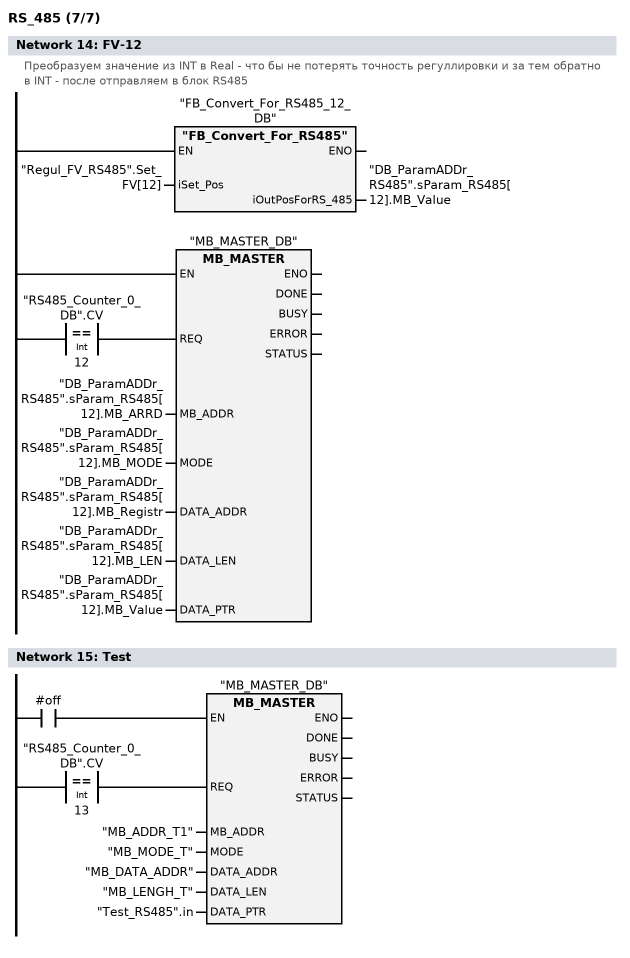
   "FB_Convert_For_RS485_12_DB"(iSet_Pos := "Regul_FV_RS485".Set_FV[12],   // "FB_Convert_For_RS485"
                           iOutPosForRS_485 => "DB_ParamADDr_RS485".sParam_RS485[12].MB_Value);
   "MB_MASTER_DB"(REQ := "RS485_Counter_0_DB".CV = 12,   // MB_MASTER
                  MB_ADDR := "DB_ParamADDr_RS485".sParam_RS485[12].MB_ARRD,
                  MODE := "DB_ParamADDr_RS485".sParam_RS485[12].MB_MODE,
                  DATA_ADDR := "DB_ParamADDr_RS485".sParam_RS485[12].MB_Registr,
                  DATA_LEN := "DB_ParamADDr_RS485".sParam_RS485[12].MB_LEN,
                  DATA_PTR := "DB_ParamADDr_RS485".sParam_RS485[12].MB_Value);
END_REGION

REGION Network 15: Test
   IF #off THEN
       "MB_MASTER_DB"(REQ := "RS485_Counter_0_DB".CV = 13,   // MB_MASTER
                      MB_ADDR := "MB_ADDR_T1",
                      MODE := "MB_MODE_T",
                      DATA_ADDR := "MB_DATA_ADDR",
                      DATA_LEN := "MB_LENGH_T",
                      DATA_PTR := "Test_RS485".in);
   END_IF;
END_REGION
END_ORGANIZATION_BLOCK

// folder: AI_Signal

FUNCTION_BLOCK "AI_(4-20)_1"   // FB13, LAD
{ S7_Optimized_Access := 'FALSE' }
VERSION : 0.1
   VAR_INPUT
      Input_PLC : Int;   // Вход_Значение на ПЛК
      "HMI_Simulate_on/off" : Bool;   // 0 - выкл, 1 - вкл
      HMI_rSimulate_value : Real;   // значение
      HMI_rParam_Sensor_HL : Real := 16.0;   // Параметры датчика по паспорту (макс значение)bar, C, итд
      HMI_rParam_Sensor_LL : Real;   // Параметры датчика по паспорту (мин значение)bar, C, итд
      "HMI_Filtr_On/off" : Bool;   // Фильтрация, true - вкл
   END_VAR
   VAR_OUTPUT
      Error_out : Bool;   // Ошибка датчика
      HMI_Value_OUT : Real;   // Значение в ед. измерения
   END_VAR
   VAR
      OUT_Scale : Real;   // Выход скалированного значения
      OUT_Normal_Ed : Real;   // Выход нормализованной единицы от 0 др 1
      AI_filtr : "AI_Filtr";
      HMI_Range : Int := 10;   // Кол-во данных для фильтрации
      HMI_iSet_Tik : Int := 2;   // Скорость набора данных для фильтрации
   END_VAR
   VAR_TEMP
      Input_PLC_to_dint : DInt;   // Конвертация из инт в реал
      Error : Word;   // Ошибка в скалировании
      "PLC to_real" : Real;
      value_scale : Real;
      Input_PLC_temp : Int;
      OFF_Param : Bool;
   END_VAR
BEGIN

REGION Network 1
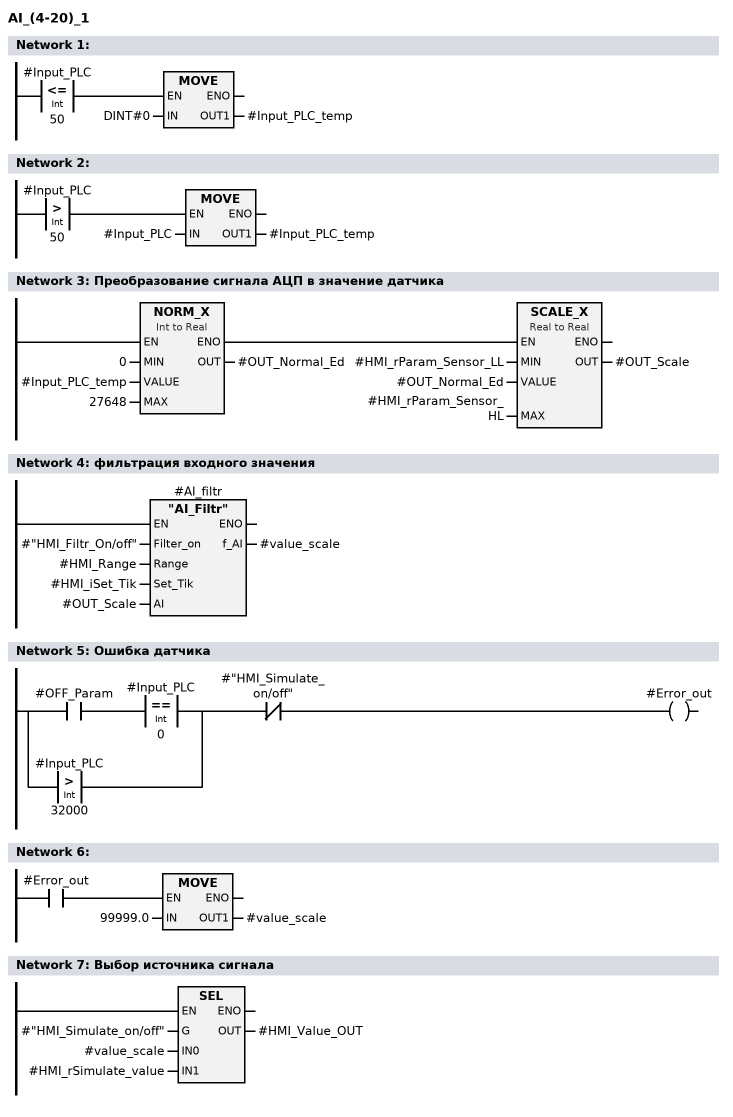
   RUNG wire#powerrail
      { S7_Templates := "SrcType := Int" } LE_Contact(in1 := #Input_PLC, in2 := 50)
      { S7_GenerateENO := "TRUE" } Move(in := DINT#0, out1 => #Input_PLC_temp)
   END_RUNG
   // the same network as SCL:
   IF #Input_PLC <= 50 THEN #Input_PLC_temp := DINT#0; END_IF;
END_REGION

REGION Network 2
   RUNG wire#powerrail
      { S7_Templates := "SrcType := Int" } GT_Contact(in1 := #Input_PLC, in2 := 50)
      { S7_GenerateENO := "TRUE" } Move(in := #Input_PLC, out1 => #Input_PLC_temp)
   END_RUNG
   // the same network as SCL:
   IF #Input_PLC > 50 THEN #Input_PLC_temp := #Input_PLC; END_IF;
END_REGION

REGION Network 3: Преобразование сигнала АЦП в значение датчика
   RUNG wire#powerrail
      { S7_Templates := "[SrcType := Int, DestType := Real]" } Normalize(min := 0, value := #Input_PLC_temp, max := 27648, out => #OUT_Normal_Ed)
      { S7_Templates := "[SrcType := Real, DestType := Real]" } Scale(min := #HMI_rParam_Sensor_LL, value := #OUT_Normal_Ed, max := #HMI_rParam_Sensor_HL, out => #OUT_Scale)
   END_RUNG
   // the same network as SCL:
   #OUT_Normal_Ed := NORM_X(MIN := 0, VALUE := #Input_PLC_temp, MAX := 27648);
   #OUT_Scale := SCALE_X(MIN := #HMI_rParam_Sensor_LL, VALUE := #OUT_Normal_Ed, MAX := #HMI_rParam_Sensor_HL);
END_REGION

REGION Network 4: фильтрация входного значения
   RUNG wire#powerrail
      #AI_filtr(Filter_on := #"HMI_Filtr_On/off", Range := #HMI_Range, Set_Tik := #HMI_iSet_Tik, AI := #OUT_Scale, f_AI => #value_scale)
   END_RUNG
   // the same network as SCL:
   #AI_filtr(Filter_on := #"HMI_Filtr_On/off",   // "AI_Filtr"
             Range := #HMI_Range,
             Set_Tik := #HMI_iSet_Tik,
             AI := #OUT_Scale,
             f_AI => #value_scale);
END_REGION

REGION Network 5: Ошибка датчика
   RUNG wire#powerrail
      Contact( #OFF_Param )
      { S7_Templates := "SrcType := Int" } EQ_Contact(in1 := #Input_PLC, in2 := 0)
      wire#w1
      I_Contact( #"HMI_Simulate_on/off" )
      Coil( #Error_out )
   END_RUNG
   RUNG wire#powerrail
      { S7_Templates := "SrcType := Int" } GT_Contact(in1 := #Input_PLC, in2 := 32000)
   END_RUNG wire#w1
   // the same network as SCL:
   #Error_out := ((#OFF_Param AND (#Input_PLC = 0)) OR (#Input_PLC > 32000)) AND NOT #"HMI_Simulate_on/off";
END_REGION

REGION Network 6
   RUNG wire#powerrail
      Contact( #Error_out )
      Move(in := 99999.0, out1 => #value_scale)
   END_RUNG
   // the same network as SCL:
   IF #Error_out THEN #value_scale := 99999.0; END_IF;
END_REGION

REGION Network 7: Выбор источника сигнала
   #HMI_Value_OUT := SEL(G := #"HMI_Simulate_on/off", IN0 := #value_scale, IN1 := #HMI_rSimulate_value);
END_REGION
END_FUNCTION_BLOCK

FUNCTION_BLOCK "AI_(PT100)"   // FB21, LAD
{ S7_Optimized_Access := 'FALSE' }
VERSION : 0.1
   VAR_INPUT
      Input_PLC : Int;   // Вход_Значение на ПЛК
      "Simulate_on/off" : Bool;   // 0 - выкл, 1 - вкл
      Simulate_value : Real;   // значение
      Param_Sensor_HL : Real := 16.0;   // Параметры датчика по паспорту (макс значение)bar, C, итд
      Param_Sensor_LL : Real;   // Параметры датчика по паспорту (мин значение)bar, C, итд
      "Filtr_On/off" : Bool;   // Фильтрация, true - вкл
   END_VAR
   VAR_OUTPUT
      Value_OUT : Real;   // Значение в ед. измерения
      Error_out : Bool;   // Ошибка датчика
   END_VAR
   VAR
      bipolar : Bool;
      OUT_Scale : Real;   // Выход скалированного значения
      AI_filtr : "AI_Filtr";
      Range : Int := 10;   // Кол-во данных для фильтрации
   END_VAR
   VAR_TEMP
      Input_PLC_to_dint : DInt;   // Конвертация из инт в реал
      Error : Word;   // Ошибка в скалировании
      "PLC to_real" : Real;
      value_scale : Real;
      Input_PLC_temp : Int;
      Input_PLC_to_real : Real;
   END_VAR
BEGIN

REGION Network 1
